TYPE "LBP_typeNC"
TITLE = NC interface / Interface CN
// User data type for block LBP_NC [DB10] / Type de données utilisateur pour bloc LBP_NC [DB10]
   STRUCT
      A_Disabl_Inp1 : Bool;   // Disable digital NCK input 1 / Bloquer entrée TOR NCK 1
      A_Disabl_Inp2 : Bool;   // Disable digital NCK input 2 / Bloquer entrée TOR NCK 2
      A_Disabl_Inp3 : Bool;   // Disable digital NCK input 3 / Bloquer entrée TOR NCK 3
      A_Disabl_Inp4 : Bool;   // Disable digital NCK input 4 / Bloquer entrée TOR NCK 4
      A_Disabl_Inp5 : Bool;   // Disable digital NCK input 5 / Bloquer entrée TOR NCK 5
      A_Disabl_Inp6 : Bool;   // Disable digital NCK input 6 / Bloquer entrée TOR NCK 6
      A_Disabl_Inp7 : Bool;   // Disable digital NCK input 7 / Bloquer entrée TOR NCK 7
      A_Disabl_Inp8 : Bool;   // Disable digital NCK input 8 / Bloquer entrée TOR NCK 8
      A_Set_Inp1 : Bool;   // Set digital NCK input 1 / Activer entrée TOR NCK 1
      A_Set_Inp2 : Bool;   // Set digital NCK input 2 / Activer entrée TOR NCK 2
      A_Set_Inp3 : Bool;   // Set digital NCK input 3 / Activer entrée TOR NCK 3
      A_Set_Inp4 : Bool;   // Set digital NCK input 4 / Activer entrée TOR NCK 4
      A_Set_Inp5 : Bool;   // Set digital NCK input 5 / Activer entrée TOR NCK 5
      A_Set_Inp6 : Bool;   // Set digital NCK input 6 / Activer entrée TOR NCK 6
      A_Set_Inp7 : Bool;   // Set digital NCK input 7 / Activer entrée TOR NCK 7
      A_Set_Inp8 : Bool;   // Set digital NCK input 8 / Activer entrée TOR NCK 8
      f0_f15 : Array[0..15] of Bool;   // Reserved / Réservé
      A_Disabl_Out1 : Bool;   // Disable digital NCK output 1 / Bloquer sortie TOR NCK 1
      A_Disabl_Out2 : Bool;   // Disable digital NCK output 2 / Bloquer sortie TOR NCK 2
      A_Disabl_Out3 : Bool;   // Disable digital NCK output 3 / Bloquer sortie TOR NCK 3
      A_Disabl_Out4 : Bool;   // Disable digital NCK output 4 / Bloquer sortie TOR NCK 4
      A_Disabl_Out5 : Bool;   // Disable digital NCK output 5 / Bloquer sortie TOR NCK 5
      A_Disabl_Out6 : Bool;   // Disable digital NCK output 6 / Bloquer sortie TOR NCK 6
      A_Disabl_Out7 : Bool;   // Disable digital NCK output 7 / Bloquer sortie TOR NCK 7
      A_Disabl_Out8 : Bool;   // Disable digital NCK output 8 / Bloquer sortie TOR NCK 8
      A_OvMask_Out1 : Bool;   // Overwrite mask of digital output 1 / Écraser le masque de sortie TOR 1
      A_OvMask_Out2 : Bool;   // Overwrite mask of digital output 2 / Écraser le masque de sortie TOR 2
      A_OvMask_Out3 : Bool;   // Overwrite mask of digital output 3 / Écraser le masque de sortie TOR 3
      A_OvMask_Out4 : Bool;   // Overwrite mask of digital output 4 / Écraser le masque de sortie TOR 4
      A_OvMask_Out5 : Bool;   // Overwrite mask of digital output 5 / Écraser le masque de sortie TOR 5
      A_OvMask_Out6 : Bool;   // Overwrite mask of digital output 6 / Écraser le masque de sortie TOR 6
      A_OvMask_Out7 : Bool;   // Overwrite mask of digital output 7 / Écraser le masque de sortie TOR 7
      A_OvMask_Out8 : Bool;   // Overwrite mask of digital output 8 / Écraser le masque de sortie TOR 8
      A_Set_Out1 : Bool;   // Set digital NCK output 1 / Activer sortie TOR NCK 1
      A_Set_Out2 : Bool;   // Set digital NCK output 2 / Activer sortie TOR NCK 2
      A_Set_Out3 : Bool;   // Set digital NCK output 3 / Activer sortie TOR NCK 3
      A_Set_Out4 : Bool;   // Set digital NCK output 4 / Activer sortie TOR NCK 4
      A_Set_Out5 : Bool;   // Set digital NCK output 5 / Activer sortie TOR NCK 5
      A_Set_Out6 : Bool;   // Set digital NCK output 6 / Activer sortie TOR NCK 6
      A_Set_Out7 : Bool;   // Set digital NCK output 7 / Activer sortie TOR NCK 7
      A_Set_Out8 : Bool;   // Set digital NCK output 8 / Activer sortie TOR NCK 8
      A_InMask_Out1 : Bool;   // Input mask of digital output 1 / Masque d'entrée de sortie TOR 1
      A_InMask_Out2 : Bool;   // Input mask of digital output 2 / Masque d'entrée de sortie TOR 2
      A_InMask_Out3 : Bool;   // Input mask of digital output 3 / Masque d'entrée de sortie TOR 3
      A_InMask_Out4 : Bool;   // Input mask of digital output 4 / Masque d'entrée de sortie TOR 4
      A_InMask_Out5 : Bool;   // Input mask of digital output 5 / Masque d'entrée de sortie TOR 5
      A_InMask_Out6 : Bool;   // Input mask of digital output 6 / Masque d'entrée de sortie TOR 6
      A_InMask_Out7 : Bool;   // Input mask of digital output 7 / Masque d'entrée de sortie TOR 7
      A_InMask_Out8 : Bool;   // Input mask of digital output 8 / Masque d'entrée de sortie TOR 8
      MCP1AxisTbl : Array[1..22] of Byte;   // Axis number Table MCP1 / Numéro d'axe table MCP1
      MCP1MaxAxis : Word;   // Max. of Axisno, must be smaller than or equal to LBP_ConfigData.MaxAxis / Le nombre max. d'axes doit être inférieur/égal à LBP_ConfigData.MaxAxis
      MCP2AxisTbl : Array[1..22] of Byte;   // Axis number Table MCP2 / Numéro d'axe table MCP2
      MCP2MaxAxis : Word;   // Max. of Axisno, must be smaller than or equal to LBP_ConfigData.MaxAxis / Le nombre max. d'axes doit être inférieur/égal à LBP_ConfigData.MaxAxis
      f56_0 : Bool;
      A_EMERGENCY : Bool;   // Emergency stop / Arrêt d'urgence
      A_EMERGENCY_Ackn : Bool;   // Acknowledge emergency stop / Acquitter arrêt d'urgence
      f56_3 : Bool;
      A_Keyswitch0 : Bool;   // Keyswitch position 0 / Position commutateur à clé 0
      A_Keyswitch1 : Bool;   // Keyswitch position 1 / Position commutateur à clé 1
      A_Keyswitch2 : Bool;   // Keyswitch position 2 / Position commutateur à clé 2
      A_Keyswitch3 : Bool;   // Keyswitch position 3 / Position commutateur à clé 3
      A_IncInModeGroup : Bool;   // INC inputs in mode group range active / Entrées INC actives dans la plage du groupe de modes de fonctionnement
      f57_1 : Bool;
      f57_2 : Bool;
      A_PCshutdown : Bool;
      f57_4 : Bool;
      f57_5 : Bool;
      A_EnableReducedDynamics : Bool;   // Enable requirement for reduced dynamics mode / Demande d'activation du mode de dynamique réduite
      f57_7 : Bool;
      A_CA_DisableAutoMach : Bool;   // Deactivate collision avoidance: AUTO Machine / Désactiver prévention des collisions : AUTO machine
      A_CA_DisableAutoTools : Bool;   // Deactivate collision avoidance: AUTO Tools / Désactiver prévention des collisions : AUTO outils
      A_CA_DisableAutoWorkh : Bool;   // Deactivate collision avoidance: AUTO Workholder / Désactiver prévention des collisions : AUTO porte-pièce
      A_CA_DisableAutoWorkp : Bool;   // Deactivate collision avoidance: AUTO Workpieces / Désactiver prévention des collisions : AUTO pièces
      A_CA_DisableJogMach : Bool;   // Deactivate collision avoidance: JOG Machine / Désactiver prévention des collisions : JOG machine
      A_CA_DisableJogTools : Bool;   // Deactivate collision avoidance: JOG Tools / Désactiver prévention des collisions : JOG outils
      A_CA_DisableJogWorkh : Bool;   // Deactivate collision avoidance: JOG Workholder / Désactiver prévention des collisions : JOG porte-pièce
      A_CA_DisableJogWorkp : Bool;   // Deactivate collision avoidance: JOG Workpieces / Désactiver prévention des collisions : JOG pièces
      f59 : Byte;
      E_ActVal_In1 : Bool;   // Actual value of digital NCK onboard input 1 / Valeur réelle de l'entrée TOR NCK intégrée 1
      E_ActVal_In2 : Bool;   // Actual value of digital NCK onboard input 2 / Valeur réelle de l'entrée TOR NCK intégrée 2
      E_ActVal_In3 : Bool;   // Actual value of digital NCK onboard input 3 / Valeur réelle de l'entrée TOR NCK intégrée 3
      E_ActVal_In4 : Bool;   // Actual value of digital NCK onboard input 4 / Valeur réelle de l'entrée TOR NCK intégrée 4
      f60_4 : Bool;
      f60_5 : Bool;
      f60_6 : Bool;
      f60_7 : Bool;
      f61_f62 : Array[61..61] of Byte;
      E_Setpoint_Out1 : Bool;   // Setpoint of digital NCK output 1 / Consigne de la sortie TOR NCK 1
      E_Setpoint_Out2 : Bool;   // Setpoint of digital NCK output 2 / Consigne de la sortie TOR NCK 2
      E_Setpoint_Out3 : Bool;   // Setpoint of digital NCK output 3 / Consigne de la sortie TOR NCK 3
      E_Setpoint_Out4 : Bool;   // Setpoint of digital NCK output 4 / Consigne de la sortie TOR NCK 4
      E_Setpoint_Out5 : Bool;   // Setpoint of digital NCK output 5 / Consigne de la sortie TOR NCK 5
      E_Setpoint_Out6 : Bool;   // Setpoint of digital NCK output 6 / Consigne de la sortie TOR NCK 6
      E_Setpoint_Out7 : Bool;   // Setpoint of digital NCK output 7 / Consigne de la sortie TOR NCK 7
      E_Setpoint_Out8 : Bool;   // Setpoint of digital NCK output 8 / Consigne de la sortie TOR NCK 8
      f65_f67 : Array[65..66] of Byte;
      E_HW1_moved : Byte;   // Handwheel 1 moved / Manivelle 1 actionnée
      E_HW2_moved : Byte;   // Handwheel 2 moved / Manivelle 2 actionnée
      E_HW3_moved : Byte;   // Handwheel 3 moved / Manivelle 3 actionnée
      E_CounterInchMetr : Byte;   // Change counter inch/metric system of units / Modifier compteur Unités métriques / anglo-saxonnes
      E_MCP1AxisValid : Bool;   // HT8: MCP1 display valid / HT8 : MCP1 Affichage valide
      E_MCP1WCS : Bool;   // HT8: MCP1 MCS / WCS / HT8 : MCP1 SCM / SCP
      f72_2 : Bool;
      f72_3 : Bool;
      f72_4 : Bool;
      f72_5 : Bool;
      f72_6 : Bool;
      E_MCP1AxKeyDisp : Bool;   // MCP1 Axis Key Displayed / MCP1 touche d'axe affichée
      E_MCP2AxisValid : Bool;   // HT8: MCP2 display valid / HT8 : MCP2 Affichage valide
      E_MCP2WCS : Bool;   // HT8: MCP2 MCS / WCS / HT8 : MCP2 SCM / SCP
      f73_2 : Bool;
      f73_3 : Bool;
      f73_4 : Bool;
      f73_5 : Bool;
      f73_6 : Bool;
      E_MCP2AxKeyDisp : Bool;   // MCP2 Axis Key Displayed / MCP2 touche d'axe affichée
      MCP1AxisFromHMI : Array[1..6] of Byte;   // Axis number from HT8 / Numéro d'axe depuis HT8
      MCP2AxisFromHMI : Array[1..6] of Byte;   // Axis number from HT8 / Numéro d'axe depuis HT8
      res86 : Word;
      res88 : Byte;
      res89 : Byte;
      epsToPlc : Byte;
      epsFromPlc : Byte;
      f92 : Byte;
      E_CA_DisableAutoMach : Bool;   // Deactivate collision avoidance: AUTO Machine / Désactiver prévention des collisions : AUTO machine
      E_CA_DisableAutoTools : Bool;   // Deactivate collision avoidance: AUTO Tools / Désactiver prévention des collisions : AUTO outils
      E_CA_DisableAutoWorkh : Bool;   // Deactivate collision avoidance: AUTO Workholder / Désactiver prévention des collisions : AUTO porte-pièce
      E_CA_DisableAutoWorkp : Bool;   // Deactivate collision avoidance: AUTO Workpieces / Désactiver prévention des collisions : AUTO pièces
      E_CA_DisableJogMach : Bool;   // Deactivate collision avoidance: JOG Machine / Désactiver prévention des collisions : JOG machine
      E_CA_DisableJogTools : Bool;   // Deactivate collision avoidance: JOG Tools / Désactiver prévention des collisions : JOG outils
      E_CA_DisableJogWorkh : Bool;   // Disable collision avoidance: JOG Workholder / Bloquer prévention des collisions : JOG porte-pièce
      E_CA_DisableJogWorkp : Bool;   // Deactivate collision avoidance: JOG Workpieces / Désactiver prévention des collisions : JOG pièces
      E_MCP1LostPackageWarn : Bool;   // Indicates an imminent disconnect of MCP 1 / Indique une déconnexion imminente du MCP 1
      E_MCP2LostPackageWarn : Bool;   // Indicates an imminent disconnect of MCP 2 / Indique une déconnexion imminente du MCP 2
      E_HTLostPackageWarn : Bool;   // Indicates an imminent disconnect of handheld terminal / Indique une déconnexion imminente du pupitre de commande portable
      E_Op1KeyLostPackageWarn : Bool;   // Indicates an imminent disconnect of direct key unit 1 / Indique une déconnexion imminente de l'unité de touches directes 1
      E_Op2KeyLostPackageWarn : Bool;   // Indicates an imminent disconnect of direct key unit 2 / Indique une déconnexion imminente de l'unité de touches directes 2
      f94_5 : Bool;
      f94_6 : Bool;
      f94_7 : Bool;
      f95 : Byte;
      E_LanguageID : Byte;   // LanguageID on HMI / ID langue de l'IHM
      E_Chan_HW1_A : Bool;   // Channel number for handwheel1 A / Numéro de canal pour manivelle 1 A
      E_Chan_HW1_B : Bool;   // Channel number for handwheel1 B / Numéro de canal pour manivelle 1 B
      E_Chan_HW1_C : Bool;   // Channel number for handwheel1 C / Numéro de canal pour manivelle 1 C
      E_Chan_HW1_D : Bool;   // Channel number for handwheel1 D / Numéro de canal pour manivelle 1 D
      f97_4 : Bool;
      f97_5 : Bool;
      f97_6 : Bool;
      f97_7 : Bool;
      E_Chan_HW2_A : Bool;   // Channel number for handwheel2 A / Numéro de canal pour manivelle 2 A
      E_Chan_HW2_B : Bool;   // Channel number for handwheel2 B / Numéro de canal pour manivelle 2 B
      E_Chan_HW2_C : Bool;   // Channel number for handwheel2 C / Numéro de canal pour manivelle 2 C
      E_Chan_HW2_D : Bool;   // Channel number for handwheel2 D / Numéro de canal pour manivelle 2 D
      f98_4 : Bool;
      f98_5 : Bool;
      f98_6 : Bool;
      f98_7 : Bool;
      E_Chan_HW3_A : Bool;   // Channel number for handwheel3 A / Numéro de canal pour manivelle 3 A
      E_Chan_HW3_B : Bool;   // Channel number for handwheel3 B / Numéro de canal pour manivelle 3 B
      E_Chan_HW3_C : Bool;   // Channel number for handwheel3 C / Numéro de canal pour manivelle 3 C
      E_Chan_HW3_D : Bool;   // Channel number for handwheel3 D / Numéro de canal pour manivelle 3 D
      f99_4 : Bool;
      f99_5 : Bool;
      f99_6 : Bool;
      f99_7 : Bool;
      E_Ax_A_HW1 : Bool;   // Axis number for handwheel1 A / Numéro d'axe pour manivelle 1 A
      E_Ax_B_HW1 : Bool;   // Axis number for handwheel1 B / Numéro d'axe pour manivelle 1 B
      E_Ax_C_HW1 : Bool;   // Axis number for handwheel1 C / Numéro d'axe pour manivelle 1 C
      E_Ax_D_HW1 : Bool;   // Axis number for handwheel1 D / Numéro d'axe pour manivelle 1 D
      E_Ax_E_HW1 : Bool;   // Axis number for handwheel1 E / Numéro d'axe pour manivelle 1 E
      E_CHW_sel1 : Bool;   // Contour handwheel selected / Manivelle de contour sélectionnée
      E_HW_sel1 : Bool;   // Handwheel selected / Manivelle sélectionnée
      E_Mach_Ax1 : Bool;   // Machine axis / Axe machine
      E_Ax_A_HW2 : Bool;   // Axis number for handwheel2 A / Numéro d'axe pour manivelle 2 A
      E_Ax_B_HW2 : Bool;   // Axis number for handwheel2 B / Numéro d'axe pour manivelle 2 B
      E_Ax_C_HW2 : Bool;   // Axis number for handwheel2 C / Numéro d'axe pour manivelle 2 C
      E_Ax_D_HW2 : Bool;   // Axis number for handwheel2 D / Numéro d'axe pour manivelle 2 D
      E_Ax_E_HW2 : Bool;   // Axis number for handwheel2 E / Numéro d'axe pour manivelle 2 E
      E_CHW_sel2 : Bool;   // Contour handwheel selected / Manivelle de contour sélectionnée
      E_HW_sel2 : Bool;   // Handwheel selected / Manivelle sélectionnée
      E_Mach_Ax2 : Bool;   // Machine axis / Axe machine
      E_Ax_A_HW3 : Bool;   // Axis number for handwheel3 A / Numéro d'axe pour manivelle 3 A
      E_Ax_B_HW3 : Bool;   // Axis number for handwheel3 B / Numéro d'axe pour manivelle 3 B
      E_Ax_C_HW3 : Bool;   // Axis number for handwheel3 C / Numéro d'axe pour manivelle 3 C
      E_Ax_D_HW3 : Bool;   // Axis number for handwheel3 D / Numéro d'axe pour manivelle 3 D
      E_Ax_E_HW3 : Bool;   // Axis number for handwheel3 E / Numéro d'axe pour manivelle 3 E
      E_CHW_sel3 : Bool;   // Contour handwheel selected / Manivelle de contour sélectionnée
      E_HW_sel3 : Bool;   // Handwheel selected / Manivelle sélectionnée
      E_Mach_Ax3 : Bool;   // Machine axis / Axe machine
      E_RemDiag : Bool;   // Remote Diagnostic / Télédiagnostic
      f103_1 : Bool;
      f103_2 : Bool;
      f103_3 : Bool;
      f103_4 : Bool;
      E_ATready : Bool;   // AT box ready / Boîte AT prête
      E_MMCTemp : Bool;   // HMI temperature limit / HMI limite température
      E_MMCBatt : Bool;   // HMI 101/102 battery alarm / HMI 101/102 alarme batterie
      E_MCP1ready : Bool;   // MCP1 ready / MCP1 prêt
      E_MCP2ready : Bool;   // MCP2 ready / MCP2 prêt
      E_HTready : Bool;   // HT ready / HT prêt
      E_Op1KeyReady : Bool;   // OP1 ready / OP1 prêt
      E_Op2KeyReady : Bool;   // OP2 ready / OP2 prêt
      f104_5 : Bool;
      E_FirstOB1 : Bool;   // This bit is on for the first OB1 cycle / Ce bit est activé pour le premier cycle OB1
      E_NCKready : Bool;   // NCK CPU ready / CPU NCK prête
      E_CancelToolCmd : Bool;   // Terminate canceled tool command / Terminer l'ordre outil abandonné
      f105_1 : Bool;
      f105_2 : Bool;
      f105_3 : Bool;
      f105_4 : Bool;
      f105_5 : Bool;
      f105_6 : Bool;
      f105_7 : Bool;
      E_CollCheckOff : Bool;   // Collisions check off / Contrôle de collision Arrêt
      E_EMERGENCY : Bool;   // EMERGENCY STOP active / ARRÊT D'URGENCE actif
      f106_2 : Bool;
      f106_3 : Bool;
      f106_4 : Bool;
      f106_5 : Bool;
      f106_6 : Bool;
      f106_7 : Bool;
      E_InspProbe1 : Bool;   // Inspection probe 1 actuated / Palpeur 1 actionné
      E_InspProbe2 : Bool;   // Inspection probe 2 actuated / Palpeur 2 actionné
      f107_2 : Bool;
      f107_3 : Bool;
      f107_4 : Bool;
      f107_5 : Bool;
      E_NCU_LinkActive : Bool;   // NCU link active / Correction NCU active
      E_SystemInchDim : Bool;   // System inch dimension / Système dimensions en inch
      f108_0 : Bool;
      E_MMC2Ready : Bool;   // MMC2-CPU ready / CPU MMC2 prête
      E_MMCMPIready : Bool;   // MMC1-CPU on MPI ready / CPU MMC1 sur MPI prête
      E_MMCBTSSready : Bool;   // MMC1-CPU on BTSS ready / CPU MMC1 sur BTSS prête
      f108_4 : Bool;
      E_DrivesInCylOp : Bool;   // Drives in cyclic operation / Entraînements en fonctionnement cyclique
      E_611Dready : Bool;
      E_NCready : Bool;
      E_NCKalarm : Bool;   // NCK alarm present / Alarme NCK présente
      f109_1 : Bool;
      f109_2 : Bool;
      f109_3 : Bool;
      A_PC_OSfault : Bool;
      E_HTempAlarm : Bool;   // Heat sink temperature alarm NCU 573 / Alarme température radiateur NCU 573
      E_ATempAlarm : Bool;   // Air temperature alarm / Alarme température de l'air
      E_BattAlarm : Bool;   // NCK battery alarm / Alarme batterie NCK
      E_SWCamMinus : Array[0..31] of Bool;   // Software cams minus [0..31] / Cames logicielles moins [0..31]
      E_SWCamPlus : Array[0..31] of Bool;   // Software cams plus [0..31] / Cames logicielles plus [0..31]
      f118_f121 : Array[0..3] of Byte;
      A_Disabl_Inp9 : Bool;   // Disable digital NCK input 9 / Bloquer entrée TOR NCK 9
      A_Disabl_Inp10 : Bool;   // Disable digital NCK input 10 / Bloquer entrée TOR NCK 10
      A_Disabl_Inp11 : Bool;   // Disable digital NCK input 11 / Bloquer entrée TOR NCK 11
      A_Disabl_Inp12 : Bool;   // Disable digital NCK input 12 / Bloquer entrée TOR NCK 12
      A_Disabl_Inp13 : Bool;   // Disable digital NCK input 13 / Bloquer entrée TOR NCK 13
      A_Disabl_Inp14 : Bool;   // Disable digital NCK input 14 / Bloquer entrée TOR NCK 14
      A_Disabl_Inp15 : Bool;   // Disable digital NCK input 15 / Bloquer entrée TOR NCK 15
      A_Disabl_Inp16 : Bool;   // Disable digital NCK input 16 / Bloquer entrée TOR NCK 16
      A_Set_Inp9 : Bool;   // Set digital NCK input 9 / Activer entrée TOR NCK 9
      A_Set_Inp10 : Bool;   // Set digital NCK input 10 / Activer entrée TOR NCK 10
      A_Set_Inp11 : Bool;   // Set digital NCK input 11 / Activer entrée TOR NCK 11
      A_Set_Inp12 : Bool;   // Set digital NCK input 12 / Activer entrée TOR NCK 12
      A_Set_Inp13 : Bool;   // Set digital NCK input 13 / Activer entrée TOR NCK 13
      A_Set_Inp14 : Bool;   // Set digital NCK input 14 / Activer entrée TOR NCK 14
      A_Set_Inp15 : Bool;   // Set digital NCK input 15 / Activer entrée TOR NCK 15
      A_Set_Inp16 : Bool;   // Set digital NCK input 16 / Activer entrée TOR NCK 16
      A_Disabl_Inp17 : Bool;   // Disable digital NCK input 17 / Bloquer entrée TOR NCK 17
      A_Disabl_Inp18 : Bool;   // Disable digital NCK input 18 / Bloquer entrée TOR NCK 18
      A_Disabl_Inp19 : Bool;   // Disable digital NCK input 19 / Bloquer entrée TOR NCK 19
      A_Disabl_Inp20 : Bool;   // Disable digital NCK input 20 / Bloquer entrée TOR NCK 20
      A_Disabl_Inp21 : Bool;   // Disable digital NCK input 21 / Bloquer entrée TOR NCK 21
      A_Disabl_Inp22 : Bool;   // Disable digital NCK input 22 / Bloquer entrée TOR NCK 22
      A_Disabl_Inp23 : Bool;   // Disable digital NCK input 23 / Bloquer entrée TOR NCK 23
      A_Disabl_Inp24 : Bool;   // Disable digital NCK input 24 / Bloquer entrée TOR NCK 24
      A_Set_Inp17 : Bool;   // Set digital NCK input 17 / Activer entrée TOR NCK 17
      A_Set_Inp18 : Bool;   // Set digital NCK input 18 / Activer entrée TOR NCK 18
      A_Set_Inp19 : Bool;   // Set digital NCK input 19 / Activer entrée TOR NCK 19
      A_Set_Inp20 : Bool;   // Set digital NCK input 20 / Activer entrée TOR NCK 20
      A_Set_Inp21 : Bool;   // Set digital NCK input 21 / Activer entrée TOR NCK 21
      A_Set_Inp22 : Bool;   // Set digital NCK input 22 / Activer entrée TOR NCK 22
      A_Set_Inp23 : Bool;   // Set digital NCK input 23 / Activer entrée TOR NCK 23
      A_Set_Inp24 : Bool;   // Set digital NCK input 24 / Activer entrée TOR NCK 24
      A_Disabl_Inp25 : Bool;   // Disable digital NCK input 25 / Bloquer entrée TOR NCK 25
      A_Disabl_Inp26 : Bool;   // Disable digital NCK input 26 / Bloquer entrée TOR NCK 26
      A_Disabl_Inp27 : Bool;   // Disable digital NCK input 27 / Bloquer entrée TOR NCK 27
      A_Disabl_Inp28 : Bool;   // Disable digital NCK input 28 / Bloquer entrée TOR NCK 28
      A_Disabl_Inp29 : Bool;   // Disable digital NCK input 29 / Bloquer entrée TOR NCK 29
      A_Disabl_Inp30 : Bool;   // Disable digital NCK input 30 / Bloquer entrée TOR NCK 30
      A_Disabl_Inp31 : Bool;   // Disable digital NCK input 31 / Bloquer entrée TOR NCK 31
      A_Disabl_Inp32 : Bool;   // Disable digital NCK input 32 / Bloquer entrée TOR NCK 32
      A_Set_Inp25 : Bool;   // Set digital NCK input 25 / Activer entrée TOR NCK 25
      A_Set_Inp26 : Bool;   // Set digital NCK input 26 / Activer entrée TOR NCK 26
      A_Set_Inp27 : Bool;   // Set digital NCK input 27 / Activer entrée TOR NCK 27
      A_Set_Inp28 : Bool;   // Set digital NCK input 28 / Activer entrée TOR NCK 28
      A_Set_Inp29 : Bool;   // Set digital NCK input 29 / Activer entrée TOR NCK 29
      A_Set_Inp30 : Bool;   // Set digital NCK input 30 / Activer entrée TOR NCK 30
      A_Set_Inp31 : Bool;   // Set digital NCK input 31 / Activer entrée TOR NCK 31
      A_Set_Inp32 : Bool;   // Set digital NCK input 32 / Activer entrée TOR NCK 32
      A_Disabl_Inp33 : Bool;   // Disable digital NCK input 33 / Bloquer entrée TOR NCK 33
      A_Disabl_Inp34 : Bool;   // Disable digital NCK input 34 / Bloquer entrée TOR NCK 34
      A_Disabl_Inp35 : Bool;   // Disable digital NCK input 35 / Bloquer entrée TOR NCK 35
      A_Disabl_Inp36 : Bool;   // Disable digital NCK input 36 / Bloquer entrée TOR NCK 36
      A_Disabl_Inp37 : Bool;   // Disable digital NCK input 37 / Bloquer entrée TOR NCK 37
      A_Disabl_Inp38 : Bool;   // Disable digital NCK input 38 / Bloquer entrée TOR NCK 38
      A_Disabl_Inp39 : Bool;   // Disable digital NCK input 39 / Bloquer entrée TOR NCK 39
      A_Disabl_Inp40 : Bool;   // Disable digital NCK input 40 / Bloquer entrée TOR NCK 40
      A_Set_Inp33 : Bool;   // Set digital NCK input 33 / Activer entrée TOR NCK 33
      A_Set_Inp34 : Bool;   // Set digital NCK input 34 / Activer entrée TOR NCK 34
      A_Set_Inp35 : Bool;   // Set digital NCK input 35 / Activer entrée TOR NCK 35
      A_Set_Inp36 : Bool;   // Set digital NCK input 36 / Activer entrée TOR NCK 36
      A_Set_Inp37 : Bool;   // Set digital NCK input 37 / Activer entrée TOR NCK 37
      A_Set_Inp38 : Bool;   // Set digital NCK input 38 / Activer entrée TOR NCK 38
      A_Set_Inp39 : Bool;   // Set digital NCK input 39 / Activer entrée TOR NCK 39
      A_Set_Inp40 : Bool;   // Set digital NCK input 40 / Activer entrée TOR NCK 40
      A_Disabl_Out9 : Bool;   // Disable digital NCK output 9 / Bloquer sortie TOR NCK 9
      A_Disabl_Out10 : Bool;   // Disable digital NCK output 10 / Bloquer sortie TOR NCK 10
      A_Disabl_Out11 : Bool;   // Disable digital NCK output 11 / Bloquer sortie TOR NCK 11
      A_Disabl_Out12 : Bool;   // Disable digital NCK output 12 / Bloquer sortie TOR NCK 12
      A_Disabl_Out13 : Bool;   // Disable digital NCK output 13 / Bloquer sortie TOR NCK 13
      A_Disabl_Out14 : Bool;   // Disable digital NCK output 14 / Bloquer sortie TOR NCK 14
      A_Disabl_Out15 : Bool;   // Disable digital NCK output 15 / Bloquer sortie TOR NCK 15
      A_Disabl_Out16 : Bool;   // Disable digital NCK output 16 / Bloquer sortie TOR NCK 16
      A_OvMask_Out9 : Bool;   // Overwrite mask of digital output 9 / Écraser le masque de sortie TOR 9
      A_OvMask_Out10 : Bool;   // Overwrite mask of digital output 10 / Écraser le masque de sortie TOR 10
      A_OvMask_Out11 : Bool;   // Overwrite mask of digital output 11 / Écraser le masque de sortie TOR 11
      A_OvMask_Out12 : Bool;   // Overwrite mask of digital output 12 / Écraser le masque de sortie TOR 12
      A_OvMask_Out13 : Bool;   // Overwrite mask of digital output 13 / Écraser le masque de sortie TOR 13
      A_OvMask_Out14 : Bool;   // Overwrite mask of digital output 14 / Écraser le masque de sortie TOR 14
      A_OvMask_Out15 : Bool;   // Overwrite mask of digital output 15 / Écraser le masque de sortie TOR 15
      A_OvMask_Out16 : Bool;   // Overwrite mask of digital output 16 / Écraser le masque de sortie TOR 16
      A_Set_Out9 : Bool;   // Set digital NCK output 9 / Activer sortie TOR NCK 9
      A_Set_Out10 : Bool;   // Set digital NCK output 10 / Activer sortie TOR NCK 10
      A_Set_Out11 : Bool;   // Set digital NCK output 11 / Activer sortie TOR NCK 11
      A_Set_Out12 : Bool;   // Set digital NCK output 12 / Activer sortie TOR NCK 12
      A_Set_Out13 : Bool;   // Set digital NCK output 13 / Activer sortie TOR NCK 13
      A_Set_Out14 : Bool;   // Set digital NCK output 14 / Activer sortie TOR NCK 14
      A_Set_Out15 : Bool;   // Set digital NCK output 15 / Activer sortie TOR NCK 15
      A_Set_Out16 : Bool;   // Set digital NCK output 16 / Activer sortie TOR NCK 16
      A_InMask_Out9 : Bool;   // Input mask of digital output 9 / Masque d'entrée de sortie TOR 9
      A_InMask_Out10 : Bool;   // Input mask of digital output 10 / Masque d'entrée de sortie TOR 10
      A_InMask_Out11 : Bool;   // Input mask of digital output 11 / Masque d'entrée de sortie TOR 11
      A_InMask_Out12 : Bool;   // Input mask of digital output 12 / Masque d'entrée de sortie TOR 12
      A_InMask_Out13 : Bool;   // Input mask of digital output 13 / Masque d'entrée de sortie TOR 13
      A_InMask_Out14 : Bool;   // Input mask of digital output 14 / Masque d'entrée de sortie TOR 14
      A_InMask_Out15 : Bool;   // Input mask of digital output 15 / Masque d'entrée de sortie TOR 15
      A_InMask_Out16 : Bool;   // Input mask of digital output 16 / Masque d'entrée de sortie TOR 16
      A_Disabl_Out17 : Bool;   // Disable digital NCK output 17 / Bloquer sortie TOR NCK 17
      A_Disabl_Out18 : Bool;   // Disable digital NCK output 18 / Bloquer sortie TOR NCK 18
      A_Disabl_Out19 : Bool;   // Disable digital NCK output 19 / Bloquer sortie TOR NCK 19
      A_Disabl_Out20 : Bool;   // Disable digital NCK output 20 / Bloquer sortie TOR NCK 20
      A_Disabl_Out21 : Bool;   // Disable digital NCK output 21 / Bloquer sortie TOR NCK 21
      A_Disabl_Out22 : Bool;   // Disable digital NCK output 22 / Bloquer sortie TOR NCK 22
      A_Disabl_Out23 : Bool;   // Disable digital NCK output 23 / Bloquer sortie TOR NCK 23
      A_Disabl_Out24 : Bool;   // Disable digital NCK output 24 / Bloquer sortie TOR NCK 24
      A_OvMask_Out17 : Bool;   // Overwrite mask of digital output 17 / Écraser le masque de sortie TOR 17
      A_OvMask_Out18 : Bool;   // Overwrite mask of digital output 18 / Écraser le masque de sortie TOR 18
      A_OvMask_Out19 : Bool;   // Overwrite mask of digital output 19 / Écraser le masque de sortie TOR 19
      A_OvMask_Out20 : Bool;   // Overwrite mask of digital output 20 / Écraser le masque de sortie TOR 20
      A_OvMask_Out21 : Bool;   // Overwrite mask of digital output 21 / Écraser le masque de sortie TOR 21
      A_OvMask_Out22 : Bool;   // Overwrite mask of digital output 22 / Écraser le masque de sortie TOR 22
      A_OvMask_Out23 : Bool;   // Overwrite mask of digital output 23 / Écraser le masque de sortie TOR 23
      A_OvMask_Out24 : Bool;   // Overwrite mask of digital output 24 / Écraser le masque de sortie TOR 24
      A_Set_Out17 : Bool;   // Set digital NCK output 17 / Activer sortie TOR NCK 17
      A_Set_Out18 : Bool;   // Set digital NCK output 18 / Activer sortie TOR NCK 18
      A_Set_Out19 : Bool;   // Set digital NCK output 19 / Activer sortie TOR NCK 19
      A_Set_Out20 : Bool;   // Set digital NCK output 20 / Activer sortie TOR NCK 20
      A_Set_Out21 : Bool;   // Set digital NCK output 21 / Activer sortie TOR NCK 21
      A_Set_Out22 : Bool;   // Set digital NCK output 22 / Activer sortie TOR NCK 22
      A_Set_Out23 : Bool;   // Set digital NCK output 23 / Activer sortie TOR NCK 23
      A_Set_Out24 : Bool;   // Set digital NCK output 24 / Activer sortie TOR NCK 24
      A_InMask_Out17 : Bool;   // Input mask of digital output 17 / Masque d'entrée de sortie TOR 17
      A_InMask_Out18 : Bool;   // Input mask of digital output 18 / Masque d'entrée de sortie TOR 18
      A_InMask_Out19 : Bool;   // Input mask of digital output 19 / Masque d'entrée de sortie TOR 19
      A_InMask_Out20 : Bool;   // Input mask of digital output 20 / Masque d'entrée de sortie TOR 20
      A_InMask_Out21 : Bool;   // Input mask of digital output 21 / Masque d'entrée de sortie TOR 21
      A_InMask_Out22 : Bool;   // Input mask of digital output 22 / Masque d'entrée de sortie TOR 22
      A_InMask_Out23 : Bool;   // Input mask of digital output 23 / Masque d'entrée de sortie TOR 23
      A_InMask_Out24 : Bool;   // Input mask of digital output 24 / Masque d'entrée de sortie TOR 24
      A_Disabl_Out25 : Bool;   // Disable digital NCK output 25 / Bloquer sortie TOR NCK 25
      A_Disabl_Out26 : Bool;   // Disable digital NCK output 26 / Bloquer sortie TOR NCK 26
      A_Disabl_Out27 : Bool;   // Disable digital NCK output 27 / Bloquer sortie TOR NCK 27
      A_Disabl_Out28 : Bool;   // Disable digital NCK output 28 / Bloquer sortie TOR NCK 28
      A_Disabl_Out29 : Bool;   // Disable digital NCK output 29 / Bloquer sortie TOR NCK 29
      A_Disabl_Out30 : Bool;   // Disable digital NCK output 30 / Bloquer sortie TOR NCK 30
      A_Disabl_Out31 : Bool;   // Disable digital NCK output 31 / Bloquer sortie TOR NCK 31
      A_Disabl_Out32 : Bool;   // Disable digital NCK output 32 / Bloquer sortie TOR NCK 32
      A_OvMask_Out25 : Bool;   // Overwrite mask of digital output 25 / Écraser le masque de sortie TOR 25
      A_OvMask_Out26 : Bool;   // Overwrite mask of digital output 26 / Écraser le masque de sortie TOR 26
      A_OvMask_Out27 : Bool;   // Overwrite mask of digital output 27 / Écraser le masque de sortie TOR 27
      A_OvMask_Out28 : Bool;   // Overwrite mask of digital output 28 / Écraser le masque de sortie TOR 28
      A_OvMask_Out29 : Bool;   // Overwrite mask of digital output 29 / Écraser le masque de sortie TOR 29
      A_OvMask_Out30 : Bool;   // Overwrite mask of digital output 30 / Écraser le masque de sortie TOR 30
      A_OvMask_Out31 : Bool;   // Overwrite mask of digital output 31 / Écraser le masque de sortie TOR 31
      A_OvMask_Out32 : Bool;   // Overwrite mask of digital output 32 / Écraser le masque de sortie TOR 32
      A_Set_Out25 : Bool;   // Set digital NCK output 25 / Activer sortie TOR NCK 25
      A_Set_Out26 : Bool;   // Set digital NCK output 26 / Activer sortie TOR NCK 26
      A_Set_Out27 : Bool;   // Set digital NCK output 27 / Activer sortie TOR NCK 27
      A_Set_Out28 : Bool;   // Set digital NCK output 28 / Activer sortie TOR NCK 28
      A_Set_Out29 : Bool;   // Set digital NCK output 29 / Activer sortie TOR NCK 29
      A_Set_Out30 : Bool;   // Set digital NCK output 30 / Activer sortie TOR NCK 30
      A_Set_Out31 : Bool;   // Set digital NCK output 31 / Activer sortie TOR NCK 31
      A_Set_Out32 : Bool;   // Set digital NCK output 32 / Activer sortie TOR NCK 32
      A_InMask_Out25 : Bool;   // Input mask of digital output 25 / Masque d'entrée de sortie TOR 25
      A_InMask_Out26 : Bool;   // Input mask of digital output 26 / Masque d'entrée de sortie TOR 26
      A_InMask_Out27 : Bool;   // Input mask of digital output 27 / Masque d'entrée de sortie TOR 27
      A_InMask_Out28 : Bool;   // Input mask of digital output 28 / Masque d'entrée de sortie TOR 28
      A_InMask_Out29 : Bool;   // Input mask of digital output 29 / Masque d'entrée de sortie TOR 29
      A_InMask_Out30 : Bool;   // Input mask of digital output 30 / Masque d'entrée de sortie TOR 30
      A_InMask_Out31 : Bool;   // Input mask of digital output 31 / Masque d'entrée de sortie TOR 31
      A_InMask_Out32 : Bool;   // Input mask of digital output 32 / Masque d'entrée de sortie TOR 32
      A_Disabl_Out33 : Bool;   // Disable digital NCK output 33 / Bloquer sortie TOR NCK 33
      A_Disabl_Out34 : Bool;   // Disable digital NCK output 34 / Bloquer sortie TOR NCK 34
      A_Disabl_Out35 : Bool;   // Disable digital NCK output 35 / Bloquer sortie TOR NCK 35
      A_Disabl_Out36 : Bool;   // Disable digital NCK output 36 / Bloquer sortie TOR NCK 36
      A_Disabl_Out37 : Bool;   // Disable digital NCK output 37 / Bloquer sortie TOR NCK 37
      A_Disabl_Out38 : Bool;   // Disable digital NCK output 38 / Bloquer sortie TOR NCK 38
      A_Disabl_Out39 : Bool;   // Disable digital NCK output 39 / Bloquer sortie TOR NCK 39
      A_Disabl_Out40 : Bool;   // Disable digital NCK output 40 / Bloquer sortie TOR NCK 40
      A_OvMask_Out33 : Bool;   // Overwrite mask of digital output 33 / Écraser le masque de sortie TOR 33
      A_OvMask_Out34 : Bool;   // Overwrite mask of digital output 34 / Écraser le masque de sortie TOR 34
      A_OvMask_Out35 : Bool;   // Overwrite mask of digital output 35 / Écraser le masque de sortie TOR 35
      A_OvMask_Out36 : Bool;   // Overwrite mask of digital output 36 / Écraser le masque de sortie TOR 36
      A_OvMask_Out37 : Bool;   // Overwrite mask of digital output 37 / Écraser le masque de sortie TOR 37
      A_OvMask_Out38 : Bool;   // Overwrite mask of digital output 38 / Écraser le masque de sortie TOR 38
      A_OvMask_Out39 : Bool;   // Overwrite mask of digital output 39 / Écraser le masque de sortie TOR 39
      A_OvMask_Out40 : Bool;   // Overwrite mask of digital output 40 / Écraser le masque de sortie TOR 40
      A_Set_Out33 : Bool;   // Set digital NCK output 33 / Activer sortie TOR NCK 33
      A_Set_Out34 : Bool;   // Set digital NCK output 34 / Activer sortie TOR NCK 34
      A_Set_Out35 : Bool;   // Set digital NCK output 35 / Activer sortie TOR NCK 35
      A_Set_Out36 : Bool;   // Set digital NCK output 36 / Activer sortie TOR NCK 36
      A_Set_Out37 : Bool;   // Set digital NCK output 37 / Activer sortie TOR NCK 37
      A_Set_Out38 : Bool;   // Set digital NCK output 38 / Activer sortie TOR NCK 38
      A_Set_Out39 : Bool;   // Set digital NCK output 39 / Activer sortie TOR NCK 39
      A_Set_Out40 : Bool;   // Set digital NCK output 40 / Activer sortie TOR NCK 40
      A_InMask_Out33 : Bool;   // Input mask of digital output 33 / Masque d'entrée de sortie TOR 33
      A_InMask_Out34 : Bool;   // Input mask of digital output 34 / Masque d'entrée de sortie TOR 34
      A_InMask_Out35 : Bool;   // Input mask of digital output 35 / Masque d'entrée de sortie TOR 35
      A_InMask_Out36 : Bool;   // Input mask of digital output 36 / Masque d'entrée de sortie TOR 36
      A_InMask_Out37 : Bool;   // Input mask of digital output 37 / Masque d'entrée de sortie TOR 37
      A_InMask_Out38 : Bool;   // Input mask of digital output 38 / Masque d'entrée de sortie TOR 38
      A_InMask_Out39 : Bool;   // Input mask of digital output 39 / Masque d'entrée de sortie TOR 39
      A_InMask_Out40 : Bool;   // Input mask of digital output 40 / Masque d'entrée de sortie TOR 40
      A_Disabl_anaIn1 : Bool;   // Disable analog NCK input 1 / Désactiver entrée analogique NCK 1
      A_Disabl_anaIn2 : Bool;   // Disable analog NCK input 2 / Désactiver entrée analogique NCK 2
      A_Disabl_anaIn3 : Bool;   // Disable analog NCK input 3 / Désactiver entrée analogique NCK 3
      A_Disabl_anaIn4 : Bool;   // Disable analog NCK input 4 / Désactiver entrée analogique NCK 4
      A_Disabl_anaIn5 : Bool;   // Disable analog NCK input 5 / Désactiver entrée analogique NCK 5
      A_Disabl_anaIn6 : Bool;   // Disable analog NCK input 6 / Désactiver entrée analogique NCK 6
      A_Disabl_anaIn7 : Bool;   // Disable analog NCK input 7 / Désactiver entrée analogique NCK 7
      A_Disabl_anaIn8 : Bool;   // Disable analog NCK input 8 / Désactiver entrée analogique NCK 8
      A_InMask_anaIn1 : Bool;   // Input mask of analog NCK input 1 / Masque d'entrée de l'entrée analogique NCK 1
      A_InMask_anaIn2 : Bool;   // Input mask of analog NCK input 2 / Masque d'entrée de l'entrée analogique NCK 2
      A_InMask_anaIn3 : Bool;   // Input mask of analog NCK input 3 / Masque d'entrée de l'entrée analogique NCK 3
      A_InMask_anaIn4 : Bool;   // Input mask of analog NCK input 4 / Masque d'entrée de l'entrée analogique NCK 4
      A_InMask_anaIn5 : Bool;   // Input mask of analog NCK input 5 / Masque d'entrée de l'entrée analogique NCK 5
      A_InMask_anaIn6 : Bool;   // Input mask of analog NCK input 6 / Masque d'entrée de l'entrée analogique NCK 6
      A_InMask_anaIn7 : Bool;   // Input mask of analog NCK input 7 / Masque d'entrée de l'entrée analogique NCK 7
      A_InMask_anaIn8 : Bool;   // Input mask of analog NCK input 8 / Masque d'entrée de l'entrée analogique NCK 8
      A_Setval_anaIn1 : Word;   // Set value of analog NCK input 1 / Activer la valeur de l'entrée analogique NCK 1
      A_Setval_anaIn2 : Word;   // Set value of analog NCK input 2 / Activer la valeur de l'entrée analogique NCK 2
      A_Setval_anaIn3 : Word;   // Set value of analog NCK input 3 / Activer la valeur de l'entrée analogique NCK 3
      A_Setval_anaIn4 : Word;   // Set value of analog NCK input 4 / Activer la valeur de l'entrée analogique NCK 4
      A_Setval_anaIn5 : Word;   // Set value of analog NCK input 5 / Activer la valeur de l'entrée analogique NCK 5
      A_Setval_anaIn6 : Word;   // Set value of analog NCK input 6 / Activer la valeur de l'entrée analogique NCK 6
      A_Setval_anaIn7 : Word;   // Set value of analog NCK input 7 / Activer la valeur de l'entrée analogique NCK 7
      A_Setval_anaIn8 : Word;   // Set value of analog NCK input 8 / Activer la valeur de l'entrée analogique NCK 8
      f164_f165 : Int;
      A_OvMask_anaOut1 : Bool;   // Overwrite mask of analog output 1 / Écraser le masque de la sortie analogique 1
      A_OvMask_anaOut2 : Bool;   // Overwrite mask of analog output 2 / Écraser le masque de la sortie analogique 2
      A_OvMask_anaOut3 : Bool;   // Overwrite mask of analog output 3 / Écraser le masque de la sortie analogique 3
      A_OvMask_anaOut4 : Bool;   // Overwrite mask of analog output 4 / Écraser le masque de la sortie analogique 4
      A_OvMask_anaOut5 : Bool;   // Overwrite mask of analog output 5 / Écraser le masque de la sortie analogique 5
      A_OvMask_anaOut6 : Bool;   // Overwrite mask of analog output 6 / Écraser le masque de la sortie analogique 6
      A_OvMask_anaOut7 : Bool;   // Overwrite mask of analog output 7 / Écraser le masque de la sortie analogique 7
      A_OvMask_anaOut8 : Bool;   // Overwrite mask of analog output 8 / Écraser le masque de la sortie analogique 8
      A_InMask_anaOut1 : Bool;   // Input mask of analog NCK output 1 / Masque d'entrée de la sortie analogique NCK 1
      A_InMask_anaOut2 : Bool;   // Input mask of analog NCK output 2 / Masque d'entrée de la sortie analogique NCK 2
      A_InMask_anaOut3 : Bool;   // Input mask of analog NCK output 3 / Masque d'entrée de la sortie analogique NCK 3
      A_InMask_anaOut4 : Bool;   // Input mask of analog NCK output 4 / Masque d'entrée de la sortie analogique NCK 4
      A_InMask_anaOut5 : Bool;   // Input mask of analog NCK output 5 / Masque d'entrée de la sortie analogique NCK 5
      A_InMask_anaOut6 : Bool;   // Input mask of analog NCK output 6 / Masque d'entrée de la sortie analogique NCK 6
      A_InMask_anaOut7 : Bool;   // Input mask of analog NCK output 7 / Masque d'entrée de la sortie analogique NCK 7
      A_InMask_anaOut8 : Bool;   // Input mask of analog NCK output 8 / Masque d'entrée de la sortie analogique NCK 8
      A_Disabl_anaOut1 : Bool;   // Disable analog NCK output 1 / Désactiver sortie analogique NCK 1
      A_Disabl_anaOut2 : Bool;   // Disable analog NCK output 2 / Désactiver sortie analogique NCK 2
      A_Disabl_anaOut3 : Bool;   // Disable analog NCK output 3 / Désactiver sortie analogique NCK 3
      A_Disabl_anaOut4 : Bool;   // Disable analog NCK output 4 / Désactiver sortie analogique NCK 4
      A_Disabl_anaOut5 : Bool;   // Disable analog NCK output 5 / Désactiver sortie analogique NCK 5
      A_Disabl_anaOut6 : Bool;   // Disable analog NCK output 6 / Désactiver sortie analogique NCK 6
      A_Disabl_anaOut7 : Bool;   // Disable analog NCK output 7 / Désactiver sortie analogique NCK 7
      A_Disabl_anaOut8 : Bool;   // Disable analog NCK output 8 / Désactiver sortie analogique NCK 8
      f169 : Byte;
      A_Setval_anaOut1 : Word;   // Set value of analog NCK output 1 / Activer la valeur de la sortie analogique NCK 1
      A_Setval_anaOut2 : Word;   // Set value of analog NCK output 2 / Activer la valeur de la sortie analogique NCK 2
      A_Setval_anaOut3 : Word;   // Set value of analog NCK output 3 / Activer la valeur de la sortie analogique NCK 3
      A_Setval_anaOut4 : Word;   // Set value of analog NCK output 4 / Activer la valeur de la sortie analogique NCK 4
      A_Setval_anaOut5 : Word;   // Set value of analog NCK output 5 / Activer la valeur de la sortie analogique NCK 5
      A_Setval_anaOut6 : Word;   // Set value of analog NCK output 6 / Activer la valeur de la sortie analogique NCK 6
      A_Setval_anaOut7 : Word;   // Set value of analog NCK output 7 / Activer la valeur de la sortie analogique NCK 7
      A_Setval_anaOut8 : Word;   // Set value of analog NCK output 8 / Activer la valeur de la sortie analogique NCK 8
      E_ActVal_In9 : Bool;   // Actual value of digital NCK input 9 / Valeur réelle de l'entrée TOR NCK 9
      E_ActVal_In10 : Bool;   // Actual value of digital NCK input 10 / Valeur réelle de l'entrée TOR NCK 10
      E_ActVal_In11 : Bool;   // Actual value of digital NCK input 11 / Valeur réelle de l'entrée TOR NCK 11
      E_ActVal_In12 : Bool;   // Actual value of digital NCK input 12 / Valeur réelle de l'entrée TOR NCK 12
      E_ActVal_In13 : Bool;   // Actual value of digital NCK input 13 / Valeur réelle de l'entrée TOR NCK 13
      E_ActVal_In14 : Bool;   // Actual value of digital NCK input 14 / Valeur réelle de l'entrée TOR NCK 14
      E_ActVal_In15 : Bool;   // Actual value of digital NCK input 15 / Valeur réelle de l'entrée TOR NCK 15
      E_ActVal_In16 : Bool;   // Actual value of digital NCK input 16 / Valeur réelle de l'entrée TOR NCK 16
      E_ActVal_In17 : Bool;   // Actual value of digital NCK input 17 / Valeur réelle de l'entrée TOR NCK 17
      E_ActVal_In18 : Bool;   // Actual value of digital NCK input 18 / Valeur réelle de l'entrée TOR NCK 18
      E_ActVal_In19 : Bool;   // Actual value of digital NCK input 19 / Valeur réelle de l'entrée TOR NCK 19
      E_ActVal_In20 : Bool;   // Actual value of digital NCK input 20 / Valeur réelle de l'entrée TOR NCK 20
      E_ActVal_In21 : Bool;   // Actual value of digital NCK input 21 / Valeur réelle de l'entrée TOR NCK 21
      E_ActVal_In22 : Bool;   // Actual value of digital NCK input 22 / Valeur réelle de l'entrée TOR NCK 22
      E_ActVal_In23 : Bool;   // Actual value of digital NCK input 23 / Valeur réelle de l'entrée TOR NCK 23
      E_ActVal_In24 : Bool;   // Actual value of digital NCK input 24 / Valeur réelle de l'entrée TOR NCK 24
      E_ActVal_In25 : Bool;   // Actual value of digital NCK input 25 / Valeur réelle de l'entrée TOR NCK 25
      E_ActVal_In26 : Bool;   // Actual value of digital NCK input 26 / Valeur réelle de l'entrée TOR NCK 26
      E_ActVal_In27 : Bool;   // Actual value of digital NCK input 27 / Valeur réelle de l'entrée TOR NCK 27
      E_ActVal_In28 : Bool;   // Actual value of digital NCK input 28 / Valeur réelle de l'entrée TOR NCK 28
      E_ActVal_In29 : Bool;   // Actual value of digital NCK input 29 / Valeur réelle de l'entrée TOR NCK 29
      E_ActVal_In30 : Bool;   // Actual value of digital NCK input 30 / Valeur réelle de l'entrée TOR NCK 30
      E_ActVal_In31 : Bool;   // Actual value of digital NCK input 31 / Valeur réelle de l'entrée TOR NCK 31
      E_ActVal_In32 : Bool;   // Actual value of digital NCK input 32 / Valeur réelle de l'entrée TOR NCK 32
      E_ActVal_In33 : Bool;   // Actual value of digital NCK input 33 / Valeur réelle de l'entrée TOR NCK 33
      E_ActVal_In34 : Bool;   // Actual value of digital NCK input 34 / Valeur réelle de l'entrée TOR NCK 34
      E_ActVal_In35 : Bool;   // Actual value of digital NCK input 35 / Valeur réelle de l'entrée TOR NCK 35
      E_ActVal_In36 : Bool;   // Actual value of digital NCK input 36 / Valeur réelle de l'entrée TOR NCK 36
      E_ActVal_In37 : Bool;   // Actual value of digital NCK input 37 / Valeur réelle de l'entrée TOR NCK 37
      E_ActVal_In38 : Bool;   // Actual value of digital NCK input 38 / Valeur réelle de l'entrée TOR NCK 38
      E_ActVal_In39 : Bool;   // Actual value of digital NCK input 39 / Valeur réelle de l'entrée TOR NCK 39
      E_ActVal_In40 : Bool;   // Actual value of digital NCK input 40 / Valeur réelle de l'entrée TOR NCK 40
      E_Setpoint_Out9 : Bool;   // Setpoint of digital NCK output 9 / Consigne de la sortie TOR NCK 9
      E_Setpoint_Out10 : Bool;   // Setpoint of digital NCK output 10 / Consigne de la sortie TOR NCK 10
      E_Setpoint_Out11 : Bool;   // Setpoint of digital NCK output 11 / Consigne de la sortie TOR NCK 11
      E_Setpoint_Out12 : Bool;   // Setpoint of digital NCK output 12 / Consigne de la sortie TOR NCK 12
      E_Setpoint_Out13 : Bool;   // Setpoint of digital NCK output 13 / Consigne de la sortie TOR NCK 13
      E_Setpoint_Out14 : Bool;   // Setpoint of digital NCK output 14 / Consigne de la sortie TOR NCK 14
      E_Setpoint_Out15 : Bool;   // Setpoint of digital NCK output 15 / Consigne de la sortie TOR NCK 15
      E_Setpoint_Out16 : Bool;   // Setpoint of digital NCK output 16 / Consigne de la sortie TOR NCK 16
      E_Setpoint_Out17 : Bool;   // Setpoint of digital NCK output 17 / Consigne de la sortie TOR NCK 17
      E_Setpoint_Out18 : Bool;   // Setpoint of digital NCK output 18 / Consigne de la sortie TOR NCK 18
      E_Setpoint_Out19 : Bool;   // Setpoint of digital NCK output 19 / Consigne de la sortie TOR NCK 19
      E_Setpoint_Out20 : Bool;   // Setpoint of digital NCK output 20 / Consigne de la sortie TOR NCK 20
      E_Setpoint_Out21 : Bool;   // Setpoint of digital NCK output 21 / Consigne de la sortie TOR NCK 21
      E_Setpoint_Out22 : Bool;   // Setpoint of digital NCK output 22 / Consigne de la sortie TOR NCK 22
      E_Setpoint_Out23 : Bool;   // Setpoint of digital NCK output 23 / Consigne de la sortie TOR NCK 23
      E_Setpoint_Out24 : Bool;   // Setpoint of digital NCK output 24 / Consigne de la sortie TOR NCK 24
      E_Setpoint_Out25 : Bool;   // Setpoint of digital NCK output 25 / Consigne de la sortie TOR NCK 25
      E_Setpoint_Out26 : Bool;   // Setpoint of digital NCK output 26 / Consigne de la sortie TOR NCK 26
      E_Setpoint_Out27 : Bool;   // Setpoint of digital NCK output 27 / Consigne de la sortie TOR NCK 27
      E_Setpoint_Out28 : Bool;   // Setpoint of digital NCK output 28 / Consigne de la sortie TOR NCK 28
      E_Setpoint_Out29 : Bool;   // Setpoint of digital NCK output 29 / Consigne de la sortie TOR NCK 29
      E_Setpoint_Out30 : Bool;   // Setpoint of digital NCK output 30 / Consigne de la sortie TOR NCK 30
      E_Setpoint_Out31 : Bool;   // Setpoint of digital NCK output 31 / Consigne de la sortie TOR NCK 31
      E_Setpoint_Out32 : Bool;   // Setpoint of digital NCK output 32 / Consigne de la sortie TOR NCK 32
      E_Setpoint_Out33 : Bool;   // Setpoint of digital NCK output 33 / Consigne de la sortie TOR NCK 33
      E_Setpoint_Out34 : Bool;   // Setpoint of digital NCK output 34 / Consigne de la sortie TOR NCK 34
      E_Setpoint_Out35 : Bool;   // Setpoint of digital NCK output 35 / Consigne de la sortie TOR NCK 35
      E_Setpoint_Out36 : Bool;   // Setpoint of digital NCK output 36 / Consigne de la sortie TOR NCK 36
      E_Setpoint_Out37 : Bool;   // Setpoint of digital NCK output 37 / Consigne de la sortie TOR NCK 37
      E_Setpoint_Out38 : Bool;   // Setpoint of digital NCK output 38 / Consigne de la sortie TOR NCK 38
      E_Setpoint_Out39 : Bool;   // Setpoint of digital NCK output 39 / Consigne de la sortie TOR NCK 39
      E_Setpoint_Out40 : Bool;   // Setpoint of digital NCK output 40 / Consigne de la sortie TOR NCK 40
      E_ActVal_anaIn1 : Word;   // Actual value of analog NCK input 1 / Valeur réelle de l'entrée analogique NCK 1
      E_ActVal_anaIn2 : Word;   // Actual value of analog NCK input 2 / Valeur réelle de l'entrée analogique NCK 2
      E_ActVal_anaIn3 : Word;   // Actual value of analog NCK input 3 / Valeur réelle de l'entrée analogique NCK 3
      E_ActVal_anaIn4 : Word;   // Actual value of analog NCK input 4 / Valeur réelle de l'entrée analogique NCK 4
      E_ActVal_anaIn5 : Word;   // Actual value of analog NCK input 5 / Valeur réelle de l'entrée analogique NCK 5
      E_ActVal_anaIn6 : Word;   // Actual value of analog NCK input 6 / Valeur réelle de l'entrée analogique NCK 6
      E_ActVal_anaIn7 : Word;   // Actual value of analog NCK input 7 / Valeur réelle de l'entrée analogique NCK 7
      E_ActVal_anaIn8 : Word;   // Actual value of analog NCK input 8 / Valeur réelle de l'entrée analogique NCK 8
      E_Setval_anaOut1 : Word;   // Set value of analog NCK output 1 / Activer la valeur de la sortie analogique NCK 1
      E_Setval_anaOut2 : Word;   // Set value of analog NCK output 2 / Activer la valeur de la sortie analogique NCK 2
      E_Setval_anaOut3 : Word;   // Set value of analog NCK output 3 / Activer la valeur de la sortie analogique NCK 3
      E_Setval_anaOut4 : Word;   // Set value of analog NCK output 4 / Activer la valeur de la sortie analogique NCK 4
      E_Setval_anaOut5 : Word;   // Set value of analog NCK output 5 / Activer la valeur de la sortie analogique NCK 5
      E_Setval_anaOut6 : Word;   // Set value of analog NCK output 6 / Activer la valeur de la sortie analogique NCK 6
      E_Setval_anaOut7 : Word;   // Set value of analog NCK output 7 / Activer la valeur de la sortie analogique NCK 7
      E_Setval_anaOut8 : Word;   // Set value of analog NCK output 8 / Activer la valeur de la sortie analogique NCK 8
      E_CollCheck : Array[0..7] of Byte;   // Collisions check / Contrôle de collision
      A_CollCheck : Array[0..7] of Byte;   // Collisions check / Contrôle de collision
      E_HW4_moved : Byte;   // Handwheel 4 moved / Manivelle 4 actionnée
      E_HW5_moved : Byte;   // Handwheel 5 moved / Manivelle 5 actionnée
      E_HW6_moved : Byte;   // Handwheel 6 moved / Manivelle 6 actionnée
      E_EHW1_stands : Bool;   // Ethernet handwheel 1 at rest / Manivelle Ethernet 1 en repos
      E_EHW2_stands : Bool;   // Ethernet handwheel 2 at rest / Manivelle Ethernet 2 en repos
      E_EHW3_stands : Bool;   // Ethernet handwheel 3 at rest / Manivelle Ethernet 3 en repos
      E_EHW4_stands : Bool;   // Ethernet handwheel 4 at rest / Manivelle Ethernet 4 en repos
      E_EHW5_stands : Bool;   // Ethernet handwheel 5 at rest / Manivelle Ethernet 5 en repos
      E_EHW6_stands : Bool;   // Ethernet handwheel 6 at rest / Manivelle Ethernet 6 en repos
      f245_6 : Bool;
      f245_7 : Bool;
      E_HMI_HW1Active : Bool;   // Handwheel 1 active / Manivelle 1 active
      E_HMI_HW2Active : Bool;   // Handwheel 2 active / Manivelle 2 active
      E_HMI_HW3Active : Bool;   // Handwheel 3 active / Manivelle 3 active
      E_HMI_HW4Active : Bool;   // Handwheel 4 active / Manivelle 4 active
      E_HMI_HW5Active : Bool;   // Handwheel 5 active / Manivelle 5 active
      E_HMI_HW6Active : Bool;   // Handwheel 6 active / Manivelle 6 active
      f246_6 : Bool;
      f246_7 : Bool;
      f247 : Byte;
      A_RobotStatus : Array[0..7] of Byte;   // Robot status / État robot
      E_RobotControl : Array[0..7] of Byte;   // Robot control / Commande de robot
   END_STRUCT;
   // MCP1AxisTbl[1] := B#16#01;
   // MCP1AxisTbl[2] := B#16#02;
   // MCP1AxisTbl[3] := B#16#03;
   // MCP1AxisTbl[4] := B#16#04;
   // MCP1AxisTbl[5] := B#16#05;
   // MCP1AxisTbl[6] := B#16#06;
   // MCP1AxisTbl[7] := B#16#07;
   // MCP1AxisTbl[8] := B#16#08;
   // MCP1AxisTbl[9] := B#16#09;
   // MCP1AxisTbl[10] := B#16#0A;
   // MCP1AxisTbl[11] := B#16#0B;
   // MCP1AxisTbl[12] := B#16#0C;
   // MCP2AxisTbl[1] := B#16#01;
   // MCP2AxisTbl[2] := B#16#02;
   // MCP2AxisTbl[3] := B#16#03;
   // MCP2AxisTbl[4] := B#16#04;
   // MCP2AxisTbl[5] := B#16#05;
   // MCP2AxisTbl[6] := B#16#06;
   // MCP2AxisTbl[7] := B#16#07;
   // MCP2AxisTbl[8] := B#16#08;
   // MCP2AxisTbl[9] := B#16#09;
   // MCP2AxisTbl[10] := B#16#0A;
   // MCP2AxisTbl[11] := B#16#0B;
   // MCP2AxisTbl[12] := B#16#0C;
END_TYPE

TYPE "LBP_typeNCKProcessIRTFlags"
TITLE = LBP_NCKProcessIRT Output Interface / LBP_NCKProcessIRT Interface sortie
// User data type for LBP_NCKProcessIRT[FC3] Output Parameters / Type de données utilisateur pour LBP_NCKProcessIRT[FC3] Paramètres de sortie
   STRUCT
      IRFromNck : Bool;   // Interrupt from NCK / Interruption en provenance du NCK
      TM : Bool;   // Tool change / Changement d'outil
      InPosition : Array[1..31] of Bool;   // Axis or spindle position reached / Position d'axe ou de broche atteinte
      AuxFunction : Array[1..10] of Bool;   // Auxiliary function available / Fonction auxiliaire disponible
   END_STRUCT;
END_TYPE

TYPE "LBP_typeTMLoad"
TITLE = Tool management / Gestion des outils
// User data type for block LBP_TMLoad [DB71] / Type de données utilisateur pour bloc LBP_TMLoad [DB71]
   STRUCT
      IFNo : Array[1..16] of Bool;   // Interface [number] active / Interface [numéro] active
      Quit : Array[1..16] of Bool;   // Perform Quit-End / Effectuer Quit-End
      TIF : Array[1..16] of Struct
         Loading : Bool;   // Loading the tool / Outil en cours de chargement
         Unloading : Bool;   // Unloading the tool / Outil en cours de déchargement
         Reloading : Bool;   // Relocating the tool / Repositionnement de l'outil
         Positioning : Bool;   // Positioning the magazine / Magasin en cours de positionnement
         PosbyProgram : Bool;   // Initiation by CNC program / Initiation par programme CNC
         PositioningMT : Bool;   // Positioning multitool / Multitool en cours de positionnement
         f0_6 : Bool;   // Reserved / Réservé
         f0_7 : Bool;   // Reserved / Réservé
         PerfStatusError : Bool;   // Negative acknowledge / Acquittement négatif
         n1_1 : Bool;   // Reserved / Réservé
         n1_2 : Bool;   // Reserved / Réservé
         n1_3 : Bool;   // Reserved / Réservé
         n1_4 : Bool;   // Reserved / Réservé
         n1_5 : Bool;   // Reserved / Réservé
         n1_6 : Bool;   // Reserved / Réservé
         DataInDB1071 : Bool;   // Multitool data stored in DB1071 / Données Multitool enregistrées dans DB1071
         Channel : Byte;   // Assigned channel / Canal affecté
         TMNo : Byte;   // Tool management number / Numéro de gestion des outils
         reserved1 : DInt;   // Reserved / Réservé
         reserved2 : DInt;   // Reserved / Réservé
         reserved3 : DInt;   // Reserved / Réservé
         LoadIdent : Int;   // Identification for loading/unloading station / Identifiant de la station de chargement/déchargement
         LoadNo : Int;   // Number of loading station / Numéro de la station de chargement
         SMag : Int;   // Magazine number (source) for unloading/reloading/pos. / Numéro de magasin (source) pour déchargement/rechargement/pos.
         SLoc : Int;   // Location number (source) for unloading/reloading/pos. / Numéro d'emplacement (source) pour déchargement/rechargement/pos.
         TMag : Int;   // Magazine number (target) for loading/reloading / Numéro de magasin (cible) pour déchargement/rechargement
         TLoc : Int;   // Location number (target) for loading/reloading / Numéro d'emplacement (cible) pour déchargement/rechargement
         WithoutMagMoving : Bool;   // HMI Data: without magazine moving / Données HMI : sans déplacement du magasin
         Res2 : Byte;   // Reserved / Réservé
      END_STRUCT;
   END_STRUCT;
   // // TIF[2].Loading : Loading the tool / Outil en cours de chargement
   // // TIF[3].Loading : Loading the tool / Outil en cours de chargement
   // // TIF[4].Loading : Loading the tool / Outil en cours de chargement
   // // TIF[5].Loading : Loading the tool / Outil en cours de chargement
   // // TIF[6].Loading : Loading the tool / Outil en cours de chargement
   // // TIF[7].Loading : Loading the tool / Outil en cours de chargement
   // // TIF[8].Loading : Loading the tool / Outil en cours de chargement
   // // TIF[9].Loading : Loading the tool / Outil en cours de chargement
   // // TIF[10].Loading : Loading the tool / Outil en cours de chargement
   // // TIF[11].Loading : Loading the tool / Outil en cours de chargement
   // // TIF[12].Loading : Loading the tool / Outil en cours de chargement
   // // TIF[13].Loading : Loading the tool / Outil en cours de chargement
   // // TIF[14].Loading : Loading the tool / Outil en cours de chargement
   // // TIF[15].Loading : Loading the tool / Outil en cours de chargement
   // // TIF[16].Loading : Loading the tool / Outil en cours de chargement
   // // TIF[2].Unloading : Unloading the tool / Outil en cours de déchargement
   // // TIF[3].Unloading : Unloading the tool / Outil en cours de déchargement
   // // TIF[4].Unloading : Unloading the tool / Outil en cours de déchargement
   // // TIF[5].Unloading : Unloading the tool / Outil en cours de déchargement
   // // TIF[6].Unloading : Unloading the tool / Outil en cours de déchargement
   // // TIF[7].Unloading : Unloading the tool / Outil en cours de déchargement
   // // TIF[8].Unloading : Unloading the tool / Outil en cours de déchargement
   // // TIF[9].Unloading : Unloading the tool / Outil en cours de déchargement
   // // TIF[10].Unloading : Unloading the tool / Outil en cours de déchargement
   // // TIF[11].Unloading : Unloading the tool / Outil en cours de déchargement
   // // TIF[12].Unloading : Unloading the tool / Outil en cours de déchargement
   // // TIF[13].Unloading : Unloading the tool / Outil en cours de déchargement
   // // TIF[14].Unloading : Unloading the tool / Outil en cours de déchargement
   // // TIF[15].Unloading : Unloading the tool / Outil en cours de déchargement
   // // TIF[16].Unloading : Unloading the tool / Outil en cours de déchargement
   // // TIF[2].Reloading : Relocating the tool / Repositionnement de l'outil
   // // TIF[3].Reloading : Relocating the tool / Repositionnement de l'outil
   // // TIF[4].Reloading : Relocating the tool / Repositionnement de l'outil
   // // TIF[5].Reloading : Relocating the tool / Repositionnement de l'outil
   // // TIF[6].Reloading : Relocating the tool / Repositionnement de l'outil
   // // TIF[7].Reloading : Relocating the tool / Repositionnement de l'outil
   // // TIF[8].Reloading : Relocating the tool / Repositionnement de l'outil
   // // TIF[9].Reloading : Relocating the tool / Repositionnement de l'outil
   // // TIF[10].Reloading : Relocating the tool / Repositionnement de l'outil
   // // TIF[11].Reloading : Relocating the tool / Repositionnement de l'outil
   // // TIF[12].Reloading : Relocating the tool / Repositionnement de l'outil
   // // TIF[13].Reloading : Relocating the tool / Repositionnement de l'outil
   // // TIF[14].Reloading : Relocating the tool / Repositionnement de l'outil
   // // TIF[15].Reloading : Relocating the tool / Repositionnement de l'outil
   // // TIF[16].Reloading : Relocating the tool / Repositionnement de l'outil
   // // TIF[2].Positioning : Positioning the magazine / Magasin en cours de positionnement
   // // TIF[3].Positioning : Positioning the magazine / Magasin en cours de positionnement
   // // TIF[4].Positioning : Positioning the magazine / Magasin en cours de positionnement
   // // TIF[5].Positioning : Positioning the magazine / Magasin en cours de positionnement
   // // TIF[6].Positioning : Positioning the magazine / Magasin en cours de positionnement
   // // TIF[7].Positioning : Positioning the magazine / Magasin en cours de positionnement
   // // TIF[8].Positioning : Positioning the magazine / Magasin en cours de positionnement
   // // TIF[9].Positioning : Positioning the magazine / Magasin en cours de positionnement
   // // TIF[10].Positioning : Positioning the magazine / Magasin en cours de positionnement
   // // TIF[11].Positioning : Positioning the magazine / Magasin en cours de positionnement
   // // TIF[12].Positioning : Positioning the magazine / Magasin en cours de positionnement
   // // TIF[13].Positioning : Positioning the magazine / Magasin en cours de positionnement
   // // TIF[14].Positioning : Positioning the magazine / Magasin en cours de positionnement
   // // TIF[15].Positioning : Positioning the magazine / Magasin en cours de positionnement
   // // TIF[16].Positioning : Positioning the magazine / Magasin en cours de positionnement
   // // TIF[2].PosbyProgram : Initiation by CNC program / Initiation par programme CNC
   // // TIF[3].PosbyProgram : Initiation by CNC program / Initiation par programme CNC
   // // TIF[4].PosbyProgram : Initiation by CNC program / Initiation par programme CNC
   // // TIF[5].PosbyProgram : Initiation by CNC program / Initiation par programme CNC
   // // TIF[6].PosbyProgram : Initiation by CNC program / Initiation par programme CNC
   // // TIF[7].PosbyProgram : Initiation by CNC program / Initiation par programme CNC
   // // TIF[8].PosbyProgram : Initiation by CNC program / Initiation par programme CNC
   // // TIF[9].PosbyProgram : Initiation by CNC program / Initiation par programme CNC
   // // TIF[10].PosbyProgram : Initiation by CNC program / Initiation par programme CNC
   // // TIF[11].PosbyProgram : Initiation by CNC program / Initiation par programme CNC
   // // TIF[12].PosbyProgram : Initiation by CNC program / Initiation par programme CNC
   // // TIF[13].PosbyProgram : Initiation by CNC program / Initiation par programme CNC
   // // TIF[14].PosbyProgram : Initiation by CNC program / Initiation par programme CNC
   // // TIF[15].PosbyProgram : Initiation by CNC program / Initiation par programme CNC
   // // TIF[16].PosbyProgram : Initiation by CNC program / Initiation par programme CNC
   // // TIF[2].PositioningMT : Positioning multitool / Multitool en cours de positionnement
   // // TIF[3].PositioningMT : Positioning multitool / Multitool en cours de positionnement
   // // TIF[4].PositioningMT : Positioning multitool / Multitool en cours de positionnement
   // // TIF[5].PositioningMT : Positioning multitool / Multitool en cours de positionnement
   // // TIF[6].PositioningMT : Positioning multitool / Multitool en cours de positionnement
   // // TIF[7].PositioningMT : Positioning multitool / Multitool en cours de positionnement
   // // TIF[8].PositioningMT : Positioning multitool / Multitool en cours de positionnement
   // // TIF[9].PositioningMT : Positioning multitool / Multitool en cours de positionnement
   // // TIF[10].PositioningMT : Positioning multitool / Multitool en cours de positionnement
   // // TIF[11].PositioningMT : Positioning multitool / Multitool en cours de positionnement
   // // TIF[12].PositioningMT : Positioning multitool / Multitool en cours de positionnement
   // // TIF[13].PositioningMT : Positioning multitool / Multitool en cours de positionnement
   // // TIF[14].PositioningMT : Positioning multitool / Multitool en cours de positionnement
   // // TIF[15].PositioningMT : Positioning multitool / Multitool en cours de positionnement
   // // TIF[16].PositioningMT : Positioning multitool / Multitool en cours de positionnement
   // // TIF[2].f0_6 : Reserved / Réservé
   // // TIF[3].f0_6 : Reserved / Réservé
   // // TIF[4].f0_6 : Reserved / Réservé
   // // TIF[5].f0_6 : Reserved / Réservé
   // // TIF[6].f0_6 : Reserved / Réservé
   // // TIF[7].f0_6 : Reserved / Réservé
   // // TIF[8].f0_6 : Reserved / Réservé
   // // TIF[9].f0_6 : Reserved / Réservé
   // // TIF[10].f0_6 : Reserved / Réservé
   // // TIF[11].f0_6 : Reserved / Réservé
   // // TIF[12].f0_6 : Reserved / Réservé
   // // TIF[13].f0_6 : Reserved / Réservé
   // // TIF[14].f0_6 : Reserved / Réservé
   // // TIF[15].f0_6 : Reserved / Réservé
   // // TIF[16].f0_6 : Reserved / Réservé
   // // TIF[2].f0_7 : Reserved / Réservé
   // // TIF[3].f0_7 : Reserved / Réservé
   // // TIF[4].f0_7 : Reserved / Réservé
   // // TIF[5].f0_7 : Reserved / Réservé
   // // TIF[6].f0_7 : Reserved / Réservé
   // // TIF[7].f0_7 : Reserved / Réservé
   // // TIF[8].f0_7 : Reserved / Réservé
   // // TIF[9].f0_7 : Reserved / Réservé
   // // TIF[10].f0_7 : Reserved / Réservé
   // // TIF[11].f0_7 : Reserved / Réservé
   // // TIF[12].f0_7 : Reserved / Réservé
   // // TIF[13].f0_7 : Reserved / Réservé
   // // TIF[14].f0_7 : Reserved / Réservé
   // // TIF[15].f0_7 : Reserved / Réservé
   // // TIF[16].f0_7 : Reserved / Réservé
   // // TIF[2].PerfStatusError : Negative acknowledge / Acquittement négatif
   // // TIF[3].PerfStatusError : Negative acknowledge / Acquittement négatif
   // // TIF[4].PerfStatusError : Negative acknowledge / Acquittement négatif
   // // TIF[5].PerfStatusError : Negative acknowledge / Acquittement négatif
   // // TIF[6].PerfStatusError : Negative acknowledge / Acquittement négatif
   // // TIF[7].PerfStatusError : Negative acknowledge / Acquittement négatif
   // // TIF[8].PerfStatusError : Negative acknowledge / Acquittement négatif
   // // TIF[9].PerfStatusError : Negative acknowledge / Acquittement négatif
   // // TIF[10].PerfStatusError : Negative acknowledge / Acquittement négatif
   // // TIF[11].PerfStatusError : Negative acknowledge / Acquittement négatif
   // // TIF[12].PerfStatusError : Negative acknowledge / Acquittement négatif
   // // TIF[13].PerfStatusError : Negative acknowledge / Acquittement négatif
   // // TIF[14].PerfStatusError : Negative acknowledge / Acquittement négatif
   // // TIF[15].PerfStatusError : Negative acknowledge / Acquittement négatif
   // // TIF[16].PerfStatusError : Negative acknowledge / Acquittement négatif
   // // TIF[2].n1_1 : Reserved / Réservé
   // // TIF[3].n1_1 : Reserved / Réservé
   // // TIF[4].n1_1 : Reserved / Réservé
   // // TIF[5].n1_1 : Reserved / Réservé
   // // TIF[6].n1_1 : Reserved / Réservé
   // // TIF[7].n1_1 : Reserved / Réservé
   // // TIF[8].n1_1 : Reserved / Réservé
   // // TIF[9].n1_1 : Reserved / Réservé
   // // TIF[10].n1_1 : Reserved / Réservé
   // // TIF[11].n1_1 : Reserved / Réservé
   // // TIF[12].n1_1 : Reserved / Réservé
   // // TIF[13].n1_1 : Reserved / Réservé
   // // TIF[14].n1_1 : Reserved / Réservé
   // // TIF[15].n1_1 : Reserved / Réservé
   // // TIF[16].n1_1 : Reserved / Réservé
   // // TIF[2].n1_2 : Reserved / Réservé
   // // TIF[3].n1_2 : Reserved / Réservé
   // // TIF[4].n1_2 : Reserved / Réservé
   // // TIF[5].n1_2 : Reserved / Réservé
   // // TIF[6].n1_2 : Reserved / Réservé
   // // TIF[7].n1_2 : Reserved / Réservé
   // // TIF[8].n1_2 : Reserved / Réservé
   // // TIF[9].n1_2 : Reserved / Réservé
   // // TIF[10].n1_2 : Reserved / Réservé
   // // TIF[11].n1_2 : Reserved / Réservé
   // // TIF[12].n1_2 : Reserved / Réservé
   // // TIF[13].n1_2 : Reserved / Réservé
   // // TIF[14].n1_2 : Reserved / Réservé
   // // TIF[15].n1_2 : Reserved / Réservé
   // // TIF[16].n1_2 : Reserved / Réservé
   // // TIF[2].n1_3 : Reserved / Réservé
   // // TIF[3].n1_3 : Reserved / Réservé
   // // TIF[4].n1_3 : Reserved / Réservé
   // // TIF[5].n1_3 : Reserved / Réservé
   // // TIF[6].n1_3 : Reserved / Réservé
   // // TIF[7].n1_3 : Reserved / Réservé
   // // TIF[8].n1_3 : Reserved / Réservé
   // // TIF[9].n1_3 : Reserved / Réservé
   // // TIF[10].n1_3 : Reserved / Réservé
   // // TIF[11].n1_3 : Reserved / Réservé
   // // TIF[12].n1_3 : Reserved / Réservé
   // // TIF[13].n1_3 : Reserved / Réservé
   // // TIF[14].n1_3 : Reserved / Réservé
   // // TIF[15].n1_3 : Reserved / Réservé
   // // TIF[16].n1_3 : Reserved / Réservé
   // // TIF[2].n1_4 : Reserved / Réservé
   // // TIF[3].n1_4 : Reserved / Réservé
   // // TIF[4].n1_4 : Reserved / Réservé
   // // TIF[5].n1_4 : Reserved / Réservé
   // // TIF[6].n1_4 : Reserved / Réservé
   // // TIF[7].n1_4 : Reserved / Réservé
   // // TIF[8].n1_4 : Reserved / Réservé
   // // TIF[9].n1_4 : Reserved / Réservé
   // // TIF[10].n1_4 : Reserved / Réservé
   // // TIF[11].n1_4 : Reserved / Réservé
   // // TIF[12].n1_4 : Reserved / Réservé
   // // TIF[13].n1_4 : Reserved / Réservé
   // // TIF[14].n1_4 : Reserved / Réservé
   // // TIF[15].n1_4 : Reserved / Réservé
   // // TIF[16].n1_4 : Reserved / Réservé
   // // TIF[2].n1_5 : Reserved / Réservé
   // // TIF[3].n1_5 : Reserved / Réservé
   // // TIF[4].n1_5 : Reserved / Réservé
   // // TIF[5].n1_5 : Reserved / Réservé
   // // TIF[6].n1_5 : Reserved / Réservé
   // // TIF[7].n1_5 : Reserved / Réservé
   // // TIF[8].n1_5 : Reserved / Réservé
   // // TIF[9].n1_5 : Reserved / Réservé
   // // TIF[10].n1_5 : Reserved / Réservé
   // // TIF[11].n1_5 : Reserved / Réservé
   // // TIF[12].n1_5 : Reserved / Réservé
   // // TIF[13].n1_5 : Reserved / Réservé
   // // TIF[14].n1_5 : Reserved / Réservé
   // // TIF[15].n1_5 : Reserved / Réservé
   // // TIF[16].n1_5 : Reserved / Réservé
   // // TIF[2].n1_6 : Reserved / Réservé
   // // TIF[3].n1_6 : Reserved / Réservé
   // // TIF[4].n1_6 : Reserved / Réservé
   // // TIF[5].n1_6 : Reserved / Réservé
   // // TIF[6].n1_6 : Reserved / Réservé
   // // TIF[7].n1_6 : Reserved / Réservé
   // // TIF[8].n1_6 : Reserved / Réservé
   // // TIF[9].n1_6 : Reserved / Réservé
   // // TIF[10].n1_6 : Reserved / Réservé
   // // TIF[11].n1_6 : Reserved / Réservé
   // // TIF[12].n1_6 : Reserved / Réservé
   // // TIF[13].n1_6 : Reserved / Réservé
   // // TIF[14].n1_6 : Reserved / Réservé
   // // TIF[15].n1_6 : Reserved / Réservé
   // // TIF[16].n1_6 : Reserved / Réservé
   // // TIF[2].DataInDB1071 : Multitool data stored in DB1071 / Données Multitool enregistrées dans DB1071
   // // TIF[3].DataInDB1071 : Multitool data stored in DB1071 / Données Multitool enregistrées dans DB1071
   // // TIF[4].DataInDB1071 : Multitool data stored in DB1071 / Données Multitool enregistrées dans DB1071
   // // TIF[5].DataInDB1071 : Multitool data stored in DB1071 / Données Multitool enregistrées dans DB1071
   // // TIF[6].DataInDB1071 : Multitool data stored in DB1071 / Données Multitool enregistrées dans DB1071
   // // TIF[7].DataInDB1071 : Multitool data stored in DB1071 / Données Multitool enregistrées dans DB1071
   // // TIF[8].DataInDB1071 : Multitool data stored in DB1071 / Données Multitool enregistrées dans DB1071
   // // TIF[9].DataInDB1071 : Multitool data stored in DB1071 / Données Multitool enregistrées dans DB1071
   // // TIF[10].DataInDB1071 : Multitool data stored in DB1071 / Données Multitool enregistrées dans DB1071
   // // TIF[11].DataInDB1071 : Multitool data stored in DB1071 / Données Multitool enregistrées dans DB1071
   // // TIF[12].DataInDB1071 : Multitool data stored in DB1071 / Données Multitool enregistrées dans DB1071
   // // TIF[13].DataInDB1071 : Multitool data stored in DB1071 / Données Multitool enregistrées dans DB1071
   // // TIF[14].DataInDB1071 : Multitool data stored in DB1071 / Données Multitool enregistrées dans DB1071
   // // TIF[15].DataInDB1071 : Multitool data stored in DB1071 / Données Multitool enregistrées dans DB1071
   // // TIF[16].DataInDB1071 : Multitool data stored in DB1071 / Données Multitool enregistrées dans DB1071
   // // TIF[2].Channel : Assigned channel / Canal affecté
   // // TIF[3].Channel : Assigned channel / Canal affecté
   // // TIF[4].Channel : Assigned channel / Canal affecté
   // // TIF[5].Channel : Assigned channel / Canal affecté
   // // TIF[6].Channel : Assigned channel / Canal affecté
   // // TIF[7].Channel : Assigned channel / Canal affecté
   // // TIF[8].Channel : Assigned channel / Canal affecté
   // // TIF[9].Channel : Assigned channel / Canal affecté
   // // TIF[10].Channel : Assigned channel / Canal affecté
   // // TIF[11].Channel : Assigned channel / Canal affecté
   // // TIF[12].Channel : Assigned channel / Canal affecté
   // // TIF[13].Channel : Assigned channel / Canal affecté
   // // TIF[14].Channel : Assigned channel / Canal affecté
   // // TIF[15].Channel : Assigned channel / Canal affecté
   // // TIF[16].Channel : Assigned channel / Canal affecté
   // // TIF[2].TMNo : Tool management number / Numéro de gestion des outils
   // // TIF[3].TMNo : Tool management number / Numéro de gestion des outils
   // // TIF[4].TMNo : Tool management number / Numéro de gestion des outils
   // // TIF[5].TMNo : Tool management number / Numéro de gestion des outils
   // // TIF[6].TMNo : Tool management number / Numéro de gestion des outils
   // // TIF[7].TMNo : Tool management number / Numéro de gestion des outils
   // // TIF[8].TMNo : Tool management number / Numéro de gestion des outils
   // // TIF[9].TMNo : Tool management number / Numéro de gestion des outils
   // // TIF[10].TMNo : Tool management number / Numéro de gestion des outils
   // // TIF[11].TMNo : Tool management number / Numéro de gestion des outils
   // // TIF[12].TMNo : Tool management number / Numéro de gestion des outils
   // // TIF[13].TMNo : Tool management number / Numéro de gestion des outils
   // // TIF[14].TMNo : Tool management number / Numéro de gestion des outils
   // // TIF[15].TMNo : Tool management number / Numéro de gestion des outils
   // // TIF[16].TMNo : Tool management number / Numéro de gestion des outils
   // // TIF[2].reserved1 : Reserved / Réservé
   // // TIF[3].reserved1 : Reserved / Réservé
   // // TIF[4].reserved1 : Reserved / Réservé
   // // TIF[5].reserved1 : Reserved / Réservé
   // // TIF[6].reserved1 : Reserved / Réservé
   // // TIF[7].reserved1 : Reserved / Réservé
   // // TIF[8].reserved1 : Reserved / Réservé
   // // TIF[9].reserved1 : Reserved / Réservé
   // // TIF[10].reserved1 : Reserved / Réservé
   // // TIF[11].reserved1 : Reserved / Réservé
   // // TIF[12].reserved1 : Reserved / Réservé
   // // TIF[13].reserved1 : Reserved / Réservé
   // // TIF[14].reserved1 : Reserved / Réservé
   // // TIF[15].reserved1 : Reserved / Réservé
   // // TIF[16].reserved1 : Reserved / Réservé
   // // TIF[2].reserved2 : Reserved / Réservé
   // // TIF[3].reserved2 : Reserved / Réservé
   // // TIF[4].reserved2 : Reserved / Réservé
   // // TIF[5].reserved2 : Reserved / Réservé
   // // TIF[6].reserved2 : Reserved / Réservé
   // // TIF[7].reserved2 : Reserved / Réservé
   // // TIF[8].reserved2 : Reserved / Réservé
   // // TIF[9].reserved2 : Reserved / Réservé
   // // TIF[10].reserved2 : Reserved / Réservé
   // // TIF[11].reserved2 : Reserved / Réservé
   // // TIF[12].reserved2 : Reserved / Réservé
   // // TIF[13].reserved2 : Reserved / Réservé
   // // TIF[14].reserved2 : Reserved / Réservé
   // // TIF[15].reserved2 : Reserved / Réservé
   // // TIF[16].reserved2 : Reserved / Réservé
   // // TIF[2].reserved3 : Reserved / Réservé
   // // TIF[3].reserved3 : Reserved / Réservé
   // // TIF[4].reserved3 : Reserved / Réservé
   // // TIF[5].reserved3 : Reserved / Réservé
   // // TIF[6].reserved3 : Reserved / Réservé
   // // TIF[7].reserved3 : Reserved / Réservé
   // // TIF[8].reserved3 : Reserved / Réservé
   // // TIF[9].reserved3 : Reserved / Réservé
   // // TIF[10].reserved3 : Reserved / Réservé
   // // TIF[11].reserved3 : Reserved / Réservé
   // // TIF[12].reserved3 : Reserved / Réservé
   // // TIF[13].reserved3 : Reserved / Réservé
   // // TIF[14].reserved3 : Reserved / Réservé
   // // TIF[15].reserved3 : Reserved / Réservé
   // // TIF[16].reserved3 : Reserved / Réservé
   // // TIF[2].LoadIdent : Identification for loading/unloading station / Identifiant de la station de chargement/déchargement
   // // TIF[3].LoadIdent : Identification for loading/unloading station / Identifiant de la station de chargement/déchargement
   // // TIF[4].LoadIdent : Identification for loading/unloading station / Identifiant de la station de chargement/déchargement
   // // TIF[5].LoadIdent : Identification for loading/unloading station / Identifiant de la station de chargement/déchargement
   // // TIF[6].LoadIdent : Identification for loading/unloading station / Identifiant de la station de chargement/déchargement
   // // TIF[7].LoadIdent : Identification for loading/unloading station / Identifiant de la station de chargement/déchargement
   // // TIF[8].LoadIdent : Identification for loading/unloading station / Identifiant de la station de chargement/déchargement
   // // TIF[9].LoadIdent : Identification for loading/unloading station / Identifiant de la station de chargement/déchargement
   // // TIF[10].LoadIdent : Identification for loading/unloading station / Identifiant de la station de chargement/déchargement
   // // TIF[11].LoadIdent : Identification for loading/unloading station / Identifiant de la station de chargement/déchargement
   // // TIF[12].LoadIdent : Identification for loading/unloading station / Identifiant de la station de chargement/déchargement
   // // TIF[13].LoadIdent : Identification for loading/unloading station / Identifiant de la station de chargement/déchargement
   // // TIF[14].LoadIdent : Identification for loading/unloading station / Identifiant de la station de chargement/déchargement
   // // TIF[15].LoadIdent : Identification for loading/unloading station / Identifiant de la station de chargement/déchargement
   // // TIF[16].LoadIdent : Identification for loading/unloading station / Identifiant de la station de chargement/déchargement
   // // TIF[2].LoadNo : Number of loading station / Numéro de la station de chargement
   // // TIF[3].LoadNo : Number of loading station / Numéro de la station de chargement
   // // TIF[4].LoadNo : Number of loading station / Numéro de la station de chargement
   // // TIF[5].LoadNo : Number of loading station / Numéro de la station de chargement
   // // TIF[6].LoadNo : Number of loading station / Numéro de la station de chargement
   // // TIF[7].LoadNo : Number of loading station / Numéro de la station de chargement
   // // TIF[8].LoadNo : Number of loading station / Numéro de la station de chargement
   // // TIF[9].LoadNo : Number of loading station / Numéro de la station de chargement
   // // TIF[10].LoadNo : Number of loading station / Numéro de la station de chargement
   // // TIF[11].LoadNo : Number of loading station / Numéro de la station de chargement
   // // TIF[12].LoadNo : Number of loading station / Numéro de la station de chargement
   // // TIF[13].LoadNo : Number of loading station / Numéro de la station de chargement
   // // TIF[14].LoadNo : Number of loading station / Numéro de la station de chargement
   // // TIF[15].LoadNo : Number of loading station / Numéro de la station de chargement
   // // TIF[16].LoadNo : Number of loading station / Numéro de la station de chargement
   // // TIF[2].SMag : Magazine number (source) for unloading/reloading/pos. / Numéro de magasin (source) pour déchargement/rechargement/pos.
   // // TIF[3].SMag : Magazine number (source) for unloading/reloading/pos. / Numéro de magasin (source) pour déchargement/rechargement/pos.
   // // TIF[4].SMag : Magazine number (source) for unloading/reloading/pos. / Numéro de magasin (source) pour déchargement/rechargement/pos.
   // // TIF[5].SMag : Magazine number (source) for unloading/reloading/pos. / Numéro de magasin (source) pour déchargement/rechargement/pos.
   // // TIF[6].SMag : Magazine number (source) for unloading/reloading/pos. / Numéro de magasin (source) pour déchargement/rechargement/pos.
   // // TIF[7].SMag : Magazine number (source) for unloading/reloading/pos. / Numéro de magasin (source) pour déchargement/rechargement/pos.
   // // TIF[8].SMag : Magazine number (source) for unloading/reloading/pos. / Numéro de magasin (source) pour déchargement/rechargement/pos.
   // // TIF[9].SMag : Magazine number (source) for unloading/reloading/pos. / Numéro de magasin (source) pour déchargement/rechargement/pos.
   // // TIF[10].SMag : Magazine number (source) for unloading/reloading/pos. / Numéro de magasin (source) pour déchargement/rechargement/pos.
   // // TIF[11].SMag : Magazine number (source) for unloading/reloading/pos. / Numéro de magasin (source) pour déchargement/rechargement/pos.
   // // TIF[12].SMag : Magazine number (source) for unloading/reloading/pos. / Numéro de magasin (source) pour déchargement/rechargement/pos.
   // // TIF[13].SMag : Magazine number (source) for unloading/reloading/pos. / Numéro de magasin (source) pour déchargement/rechargement/pos.
   // // TIF[14].SMag : Magazine number (source) for unloading/reloading/pos. / Numéro de magasin (source) pour déchargement/rechargement/pos.
   // // TIF[15].SMag : Magazine number (source) for unloading/reloading/pos. / Numéro de magasin (source) pour déchargement/rechargement/pos.
   // // TIF[16].SMag : Magazine number (source) for unloading/reloading/pos. / Numéro de magasin (source) pour déchargement/rechargement/pos.
   // // TIF[2].SLoc : Location number (source) for unloading/reloading/pos. / Numéro d'emplacement (source) pour déchargement/rechargement/pos.
   // // TIF[3].SLoc : Location number (source) for unloading/reloading/pos. / Numéro d'emplacement (source) pour déchargement/rechargement/pos.
   // // TIF[4].SLoc : Location number (source) for unloading/reloading/pos. / Numéro d'emplacement (source) pour déchargement/rechargement/pos.
   // // TIF[5].SLoc : Location number (source) for unloading/reloading/pos. / Numéro d'emplacement (source) pour déchargement/rechargement/pos.
   // // TIF[6].SLoc : Location number (source) for unloading/reloading/pos. / Numéro d'emplacement (source) pour déchargement/rechargement/pos.
   // // TIF[7].SLoc : Location number (source) for unloading/reloading/pos. / Numéro d'emplacement (source) pour déchargement/rechargement/pos.
   // // TIF[8].SLoc : Location number (source) for unloading/reloading/pos. / Numéro d'emplacement (source) pour déchargement/rechargement/pos.
   // // TIF[9].SLoc : Location number (source) for unloading/reloading/pos. / Numéro d'emplacement (source) pour déchargement/rechargement/pos.
   // // TIF[10].SLoc : Location number (source) for unloading/reloading/pos. / Numéro d'emplacement (source) pour déchargement/rechargement/pos.
   // // TIF[11].SLoc : Location number (source) for unloading/reloading/pos. / Numéro d'emplacement (source) pour déchargement/rechargement/pos.
   // // TIF[12].SLoc : Location number (source) for unloading/reloading/pos. / Numéro d'emplacement (source) pour déchargement/rechargement/pos.
   // // TIF[13].SLoc : Location number (source) for unloading/reloading/pos. / Numéro d'emplacement (source) pour déchargement/rechargement/pos.
   // // TIF[14].SLoc : Location number (source) for unloading/reloading/pos. / Numéro d'emplacement (source) pour déchargement/rechargement/pos.
   // // TIF[15].SLoc : Location number (source) for unloading/reloading/pos. / Numéro d'emplacement (source) pour déchargement/rechargement/pos.
   // // TIF[16].SLoc : Location number (source) for unloading/reloading/pos. / Numéro d'emplacement (source) pour déchargement/rechargement/pos.
   // // TIF[2].TMag : Magazine number (target) for loading/reloading / Numéro de magasin (cible) pour déchargement/rechargement
   // // TIF[3].TMag : Magazine number (target) for loading/reloading / Numéro de magasin (cible) pour déchargement/rechargement
   // // TIF[4].TMag : Magazine number (target) for loading/reloading / Numéro de magasin (cible) pour déchargement/rechargement
   // // TIF[5].TMag : Magazine number (target) for loading/reloading / Numéro de magasin (cible) pour déchargement/rechargement
   // // TIF[6].TMag : Magazine number (target) for loading/reloading / Numéro de magasin (cible) pour déchargement/rechargement
   // // TIF[7].TMag : Magazine number (target) for loading/reloading / Numéro de magasin (cible) pour déchargement/rechargement
   // // TIF[8].TMag : Magazine number (target) for loading/reloading / Numéro de magasin (cible) pour déchargement/rechargement
   // // TIF[9].TMag : Magazine number (target) for loading/reloading / Numéro de magasin (cible) pour déchargement/rechargement
   // // TIF[10].TMag : Magazine number (target) for loading/reloading / Numéro de magasin (cible) pour déchargement/rechargement
   // // TIF[11].TMag : Magazine number (target) for loading/reloading / Numéro de magasin (cible) pour déchargement/rechargement
   // // TIF[12].TMag : Magazine number (target) for loading/reloading / Numéro de magasin (cible) pour déchargement/rechargement
   // // TIF[13].TMag : Magazine number (target) for loading/reloading / Numéro de magasin (cible) pour déchargement/rechargement
   // // TIF[14].TMag : Magazine number (target) for loading/reloading / Numéro de magasin (cible) pour déchargement/rechargement
   // // TIF[15].TMag : Magazine number (target) for loading/reloading / Numéro de magasin (cible) pour déchargement/rechargement
   // // TIF[16].TMag : Magazine number (target) for loading/reloading / Numéro de magasin (cible) pour déchargement/rechargement
   // // TIF[2].TLoc : Location number (target) for loading/reloading / Numéro d'emplacement (cible) pour déchargement/rechargement
   // // TIF[3].TLoc : Location number (target) for loading/reloading / Numéro d'emplacement (cible) pour déchargement/rechargement
   // // TIF[4].TLoc : Location number (target) for loading/reloading / Numéro d'emplacement (cible) pour déchargement/rechargement
   // // TIF[5].TLoc : Location number (target) for loading/reloading / Numéro d'emplacement (cible) pour déchargement/rechargement
   // // TIF[6].TLoc : Location number (target) for loading/reloading / Numéro d'emplacement (cible) pour déchargement/rechargement
   // // TIF[7].TLoc : Location number (target) for loading/reloading / Numéro d'emplacement (cible) pour déchargement/rechargement
   // // TIF[8].TLoc : Location number (target) for loading/reloading / Numéro d'emplacement (cible) pour déchargement/rechargement
   // // TIF[9].TLoc : Location number (target) for loading/reloading / Numéro d'emplacement (cible) pour déchargement/rechargement
   // // TIF[10].TLoc : Location number (target) for loading/reloading / Numéro d'emplacement (cible) pour déchargement/rechargement
   // // TIF[11].TLoc : Location number (target) for loading/reloading / Numéro d'emplacement (cible) pour déchargement/rechargement
   // // TIF[12].TLoc : Location number (target) for loading/reloading / Numéro d'emplacement (cible) pour déchargement/rechargement
   // // TIF[13].TLoc : Location number (target) for loading/reloading / Numéro d'emplacement (cible) pour déchargement/rechargement
   // // TIF[14].TLoc : Location number (target) for loading/reloading / Numéro d'emplacement (cible) pour déchargement/rechargement
   // // TIF[15].TLoc : Location number (target) for loading/reloading / Numéro d'emplacement (cible) pour déchargement/rechargement
   // // TIF[16].TLoc : Location number (target) for loading/reloading / Numéro d'emplacement (cible) pour déchargement/rechargement
   // // TIF[2].WithoutMagMoving : HMI Data: without magazine moving / Données HMI : sans déplacement du magasin
   // // TIF[3].WithoutMagMoving : HMI Data: without magazine moving / Données HMI : sans déplacement du magasin
   // // TIF[4].WithoutMagMoving : HMI Data: without magazine moving / Données HMI : sans déplacement du magasin
   // // TIF[5].WithoutMagMoving : HMI Data: without magazine moving / Données HMI : sans déplacement du magasin
   // // TIF[6].WithoutMagMoving : HMI Data: without magazine moving / Données HMI : sans déplacement du magasin
   // // TIF[7].WithoutMagMoving : HMI Data: without magazine moving / Données HMI : sans déplacement du magasin
   // // TIF[8].WithoutMagMoving : HMI Data: without magazine moving / Données HMI : sans déplacement du magasin
   // // TIF[9].WithoutMagMoving : HMI Data: without magazine moving / Données HMI : sans déplacement du magasin
   // // TIF[10].WithoutMagMoving : HMI Data: without magazine moving / Données HMI : sans déplacement du magasin
   // // TIF[11].WithoutMagMoving : HMI Data: without magazine moving / Données HMI : sans déplacement du magasin
   // // TIF[12].WithoutMagMoving : HMI Data: without magazine moving / Données HMI : sans déplacement du magasin
   // // TIF[13].WithoutMagMoving : HMI Data: without magazine moving / Données HMI : sans déplacement du magasin
   // // TIF[14].WithoutMagMoving : HMI Data: without magazine moving / Données HMI : sans déplacement du magasin
   // // TIF[15].WithoutMagMoving : HMI Data: without magazine moving / Données HMI : sans déplacement du magasin
   // // TIF[16].WithoutMagMoving : HMI Data: without magazine moving / Données HMI : sans déplacement du magasin
   // // TIF[2].Res2 : Reserved / Réservé
   // // TIF[3].Res2 : Reserved / Réservé
   // // TIF[4].Res2 : Reserved / Réservé
   // // TIF[5].Res2 : Reserved / Réservé
   // // TIF[6].Res2 : Reserved / Réservé
   // // TIF[7].Res2 : Reserved / Réservé
   // // TIF[8].Res2 : Reserved / Réservé
   // // TIF[9].Res2 : Reserved / Réservé
   // // TIF[10].Res2 : Reserved / Réservé
   // // TIF[11].Res2 : Reserved / Réservé
   // // TIF[12].Res2 : Reserved / Réservé
   // // TIF[13].Res2 : Reserved / Réservé
   // // TIF[14].Res2 : Reserved / Réservé
   // // TIF[15].Res2 : Reserved / Réservé
   // // TIF[16].Res2 : Reserved / Réservé
END_TYPE

